C09107=1044.224,228.789,397.774,171.384,39.330,157.455
C09108=1044.218,228.541,397.802,171.382,39.328,157.454
C09109=1044.211,228.292,397.829,171.380,39.325,157.454
C09110=1044.204,228.044,397.856,171.378,39.323,157.453
C09111=1044.197,227.795,397.883,171.375,39.321,157.453
C09112=1044.191,227.547,397.911,171.373,39.319,157.452
C09113=1044.184,227.299,397.939,171.370,39.316,157.452
C09114=1044.178,227.051,397.966,171.369,39.314,157.451
C09115=1044.171,226.802,397.994,171.366,39.312,157.451
C09116=1044.164,226.554,398.022,171.364,39.309,157.450
C09117=1044.158,226.305,398.049,171.361,39.306,157.449
C09118=1044.151,226.056,398.076,171.358,39.304,157.449
C09119=1044.145,225.809,398.103,171.357,39.302,157.448
C09120=1044.138,225.560,398.131,171.354,39.299,157.448
C09121=1044.131,225.312,398.159,171.352,39.297,157.447
C09122=1044.125,225.063,398.186,171.349,39.295,157.446
C09123=1044.118,224.814,398.213,171.347,39.292,157.446
C09124=1044.111,224.566,398.241,171.345,39.290,157.445
C09125=1044.106,224.318,398.268,171.343,39.287,157.445
C09126=1044.099,224.069,398.296,171.340,39.285,157.444
C09127=1044.092,223.821,398.323,171.337,39.283,157.444
C09128=1044.085,223.573,398.350,171.336,39.280,157.443
C09129=1044.079,223.324,398.377,171.333,39.277,157.442
C09130=1044.072,223.076,398.405,171.331,39.275,157.442
C09131=1044.066,222.827,398.433,171.328,39.273,157.441
C09132=1044.059,222.578,398.460,171.327,39.271,157.441
C09133=1044.053,222.331,398.487,171.324,39.268,157.440
C09134=1044.046,222.082,398.514,171.322,39.266,157.440
C09135=1044.040,221.833,398.541,171.319,39.263,157.439
C09136=1044.033,221.585,398.569,171.317,39.261,157.438
C09137=1044.027,221.337,398.595,171.315,39.258,157.438
C09138=1044.019,221.044,398.628,171.312,39.255,157.437
C09139=1044.012,220.752,398.660,171.310,39.253,157.436
C09140=1044.003,220.459,398.692,171.307,39.250,157.436
C09141=1043.996,220.167,398.724,171.304,39.247,157.435
C09142=1043.990,219.918,398.751,171.302,39.244,157.434
C09143=1043.983,219.670,398.778,171.299,39.242,157.434
C09144=1043.976,219.421,398.805,171.298,39.240,157.433
C09145=1043.969,219.173,398.832,171.295,39.237,157.433
C09146=1043.963,218.925,398.859,171.293,39.235,157.432
C09147=1043.956,218.676,398.886,171.290,39.233,157.432
C09148=1043.950,218.428,398.913,171.288,39.230,157.431
C09149=1043.943,218.179,398.940,171.286,39.228,157.430
C09150=1043.936,217.930,398.966,171.283,39.225,157.430
C09151=1043.929,217.682,398.994,171.282,39.223,157.429
C09152=1043.924,217.433,399.021,171.279,39.221,157.429
C09153=1043.916,217.185,399.048,171.277,39.218,157.428
C09154=1043.910,216.936,399.075,171.275,39.216,157.428
C09155=1043.903,216.688,399.101,171.273,39.213,157.427
C09156=1043.897,216.440,399.129,171.270,39.211,157.426
C09157=1043.890,216.191,399.155,171.268,39.208,157.426
C09158=1043.884,215.943,399.182,171.266,39.206,157.425
C09159=1043.877,215.694,399.210,171.263,39.204,157.425
C09160=1043.870,215.445,399.236,171.261,39.201,157.424
C09161=1043.864,215.197,399.263,171.259,39.199,157.424
C09162=1043.857,214.949,399.290,171.257,39.196,157.423
C09163=1043.851,214.701,399.316,171.254,39.194,157.422
C09164=1043.844,214.452,399.343,171.253,39.191,157.422
C09165=1043.838,214.203,399.370,171.250,39.189,157.421
C09166=1043.829,213.866,399.406,171.247,39.186,157.420
C09167=1043.820,213.528,399.442,171.245,39.182,157.420
C09168=1043.811,213.191,399.479,171.241,39.179,157.419
C09169=1043.802,212.853,399.515,171.238,39.176,157.418
C09170=1043.796,212.606,399.542,171.237,39.173,157.418
C09171=1043.789,212.357,399.569,171.234,39.171,157.417
C09172=1043.782,212.108,399.596,171.231,39.168,157.416
C09173=1043.777,211.860,399.622,171.230,39.166,157.416
C09174=1043.769,211.611,399.649,171.227,39.163,157.415
C09175=1043.763,211.363,399.675,171.226,39.161,157.415
C09176=1043.757,211.114,399.702,171.223,39.159,157.414
C09177=1043.750,210.866,399.729,171.221,39.156,157.414
C09178=1043.743,210.617,399.756,171.219,39.153,157.413
C09179=1043.736,210.368,399.782,171.217,39.151,157.412
C09180=1043.730,210.120,399.808,171.214,39.149,157.412
C09181=1043.723,209.871,399.835,171.213,39.146,157.411
C09182=1043.717,209.623,399.861,171.210,39.144,157.411
C09183=1043.710,209.374,399.888,171.208,39.141,157.410
C09184=1043.704,209.126,399.914,171.206,39.139,157.409
C09185=1043.697,208.877,399.941,171.203,39.137,157.409
C09186=1043.690,208.629,399.967,171.202,39.134,157.408
C09187=1043.684,208.380,399.994,171.199,39.132,157.408
C09188=1043.677,208.132,400.020,171.198,39.129,157.407
C09189=1043.670,207.883,400.046,171.195,39.127,157.407
C09190=1043.665,207.660,400.071,171.194,39.125,157.406
C09191=1043.659,207.437,400.094,171.191,39.122,157.406
C09192=1043.653,207.214,400.117,171.190,39.120,157.405
C09193=1043.646,206.990,400.141,171.187,39.118,157.405
C09194=1043.641,206.767,400.164,171.186,39.116,157.404
C09195=1043.635,206.544,400.188,171.184,39.114,157.404
C09196=1043.628,206.321,400.212,171.182,39.111,157.403
C09197=1043.623,206.097,400.236,171.181,39.110,157.403
C09198=1043.597,205.046,400.342,170.913,39.008,157.374
C09199=1043.591,204.797,400.367,170.910,39.006,157.373
C09200=1043.585,204.548,400.392,170.907,39.004,157.373
C09201=1043.578,204.300,400.417,170.905,39.003,157.373
C09202=1043.572,204.051,400.442,170.901,39.001,157.372
C09203=1043.566,203.802,400.468,170.899,38.999,157.372
C09204=1043.560,203.554,400.493,170.895,38.998,157.371
C09205=1043.554,203.305,400.517,170.893,38.996,157.371
C09206=1043.548,203.056,400.543,170.890,38.994,157.370
C09207=1043.542,202.808,400.568,170.887,38.993,157.370
C09208=1043.536,202.559,400.593,170.884,38.991,157.370
C09209=1043.530,202.310,400.618,170.882,38.989,157.369
C09210=1043.524,202.062,400.643,170.879,38.987,157.369
C09211=1043.518,201.813,400.668,170.876,38.986,157.368
C09212=1043.512,201.565,400.694,170.873,38.984,157.368
C09213=1043.506,201.315,400.718,170.870,38.982,157.368
C09214=1043.499,201.067,400.743,170.868,38.981,157.367
C09215=1043.493,200.818,400.768,170.864,38.979,157.367
C09216=1043.487,200.570,400.792,170.862,38.978,157.366
C09217=1043.480,200.321,400.817,170.859,38.976,157.366
C09218=1043.474,200.072,400.842,170.856,38.975,157.366
C09219=1043.468,199.824,400.867,170.853,38.973,157.365
C09220=1043.462,199.574,400.891,170.851,38.972,157.365
C09221=1043.455,199.326,400.916,170.848,38.970,157.364
C09222=1043.449,199.077,400.940,170.845,38.968,157.364
C09223=1043.443,198.829,400.966,170.842,38.967,157.364
C09224=1043.437,198.580,400.990,170.839,38.966,157.363
C09225=1043.430,198.331,401.015,170.837,38.964,157.363
C09226=1043.424,198.082,401.039,170.833,38.962,157.362
C09227=1043.418,197.834,401.064,170.831,38.961,157.362
C09228=1043.411,197.585,401.088,170.828,38.960,157.362
C09229=1043.405,197.336,401.113,170.825,38.958,157.361
C09230=1043.399,197.087,401.138,170.823,38.956,157.361
C09231=1043.393,196.840,401.162,170.820,38.954,157.360
C09232=1043.387,196.590,401.187,170.817,38.953,157.360
C09233=1043.380,196.341,401.211,170.814,38.952,157.360
C09234=1043.374,196.093,401.236,170.812,38.950,157.359
C09235=1043.368,195.844,401.260,170.809,38.949,157.359
C09236=1043.362,195.596,401.285,170.806,38.947,157.359
C09237=1043.356,195.346,401.310,170.804,38.945,157.358
C09238=1043.350,195.098,401.334,170.800,38.944,157.358
C09239=1043.344,194.849,401.359,170.798,38.943,157.357
C09240=1043.337,194.600,401.383,170.795,38.941,157.357
C09241=1043.331,194.351,401.408,170.792,38.939,157.357
C09242=1043.325,194.104,401.432,170.790,38.938,157.356
C09243=1043.319,193.854,401.457,170.786,38.937,157.356
C09244=1043.312,193.605,401.481,170.784,38.935,157.355
C09245=1043.307,193.357,401.506,170.782,38.934,157.355
C09246=1043.301,193.108,401.530,170.778,38.932,157.355
C09247=1043.295,192.860,401.554,170.776,38.930,157.354
C09248=1043.289,192.610,401.579,170.774,38.929,157.354
C09249=1043.282,192.362,401.603,170.770,38.928,157.354
C09250=1043.277,192.113,401.628,170.768,38.926,157.353
C09251=1043.270,191.864,401.652,170.765,38.925,157.353
C09252=1043.264,191.615,401.676,170.762,38.923,157.352
C09253=1043.258,191.367,401.700,170.760,38.921,157.352
C09254=1043.252,191.118,401.725,170.757,38.920,157.352
C09255=1043.246,190.870,401.749,170.754,38.919,157.351
C09256=1043.240,190.621,401.774,170.752,38.917,157.351
C09257=1043.233,190.372,401.798,170.749,38.916,157.351
C09258=1043.228,190.123,401.822,170.746,38.914,157.350
C09259=1043.221,189.839,401.850,170.743,38.912,157.350
C09260=1043.214,189.554,401.877,170.741,38.911,157.349
C09261=1043.207,189.271,401.905,170.737,38.909,157.349
C09262=1043.201,188.985,401.933,170.734,38.907,157.349
C09263=1043.194,188.736,401.957,170.732,38.906,157.348
C09264=1043.189,188.488,401.981,170.729,38.905,157.348
C09265=1043.182,188.239,402.005,170.727,38.903,157.347
C09266=1043.176,187.991,402.030,170.724,38.902,157.347
C09267=1043.170,187.742,402.054,170.721,38.900,157.347
C09268=1043.165,187.493,402.078,170.719,38.899,157.346
C09269=1043.158,187.244,402.103,170.716,38.897,157.346
C09270=1043.153,186.996,402.127,170.713,38.895,157.346
C09271=1043.146,186.747,402.151,170.711,38.894,157.345
C09272=1043.141,186.498,402.175,170.708,38.893,157.345
C09273=1043.134,186.249,402.199,170.705,38.892,157.345
C09274=1043.129,186.001,402.223,170.703,38.890,157.344
C09275=1043.123,185.752,402.247,170.701,38.888,157.344
C09276=1043.117,185.503,402.272,170.697,38.887,157.343
C09277=1043.111,185.255,402.295,170.695,38.885,157.343
C09278=1043.104,185.005,402.319,170.693,38.884,157.343
C09279=1043.099,184.757,402.343,170.690,38.882,157.342
C09280=1043.092,184.508,402.367,170.687,38.881,157.342
C09281=1043.087,184.259,402.391,170.685,38.880,157.342
C09282=1043.081,184.010,402.415,170.682,38.878,157.341
C09283=1043.075,183.761,402.439,170.680,38.877,157.341
C09284=1043.069,183.513,402.463,170.677,38.875,157.340
C09285=1043.063,183.264,402.486,170.674,38.874,157.340
C09286=1043.056,183.015,402.510,170.672,38.873,157.340
C09287=1043.050,182.766,402.534,170.669,38.872,157.340
C09288=1043.044,182.517,402.558,170.666,38.870,157.339
C09289=1043.038,182.268,402.581,170.664,38.869,157.339
C09290=1043.031,182.019,402.605,170.661,38.868,157.339
C09291=1043.024,181.771,402.628,170.659,38.866,157.338
C09292=1043.018,181.522,402.651,170.656,38.865,157.338
C09293=1043.012,181.274,402.675,170.653,38.864,157.338
C09294=1043.005,181.025,402.699,170.651,38.863,157.337
C09295=1043.000,180.776,402.722,170.648,38.861,157.337
C09296=1042.993,180.527,402.746,170.646,38.860,157.337
C09297=1042.987,180.278,402.770,170.643,38.859,157.336
C09298=1042.981,180.030,402.793,170.641,38.858,157.336
C09299=1042.975,179.781,402.817,170.638,38.856,157.336
C09300=1042.969,179.532,402.840,170.635,38.855,157.335
C09301=1042.962,179.283,402.864,170.633,38.854,157.335
C09302=1042.957,179.034,402.887,170.631,38.853,157.335
C09303=1042.949,178.785,402.910,170.628,38.851,157.334
C09304=1042.943,178.537,402.934,170.625,38.850,157.334
C09305=1042.937,178.288,402.957,170.623,38.849,157.334
C09306=1042.931,178.039,402.981,170.620,38.848,157.334
C09307=1042.925,177.790,403.004,170.618,38.846,157.333
C09308=1042.918,177.541,403.028,170.615,38.845,157.333
C09309=1042.913,177.292,403.051,170.613,38.844,157.333
C09310=1042.907,177.044,403.074,170.610,38.843,157.332
C09311=1042.900,176.794,403.098,170.608,38.841,157.332
C09312=1042.894,176.546,403.121,170.605,38.840,157.332
C09313=1042.887,176.297,403.144,170.602,38.839,157.331
C09314=1042.881,176.049,403.168,170.600,38.838,157.331
C09315=1042.875,175.800,403.191,170.598,38.837,157.331
C09316=1042.869,175.550,403.214,170.596,38.835,157.330
C09317=1042.863,175.302,403.238,170.592,38.834,157.330
C09318=1042.857,175.053,403.261,170.590,38.833,157.330
C09319=1042.851,174.804,403.285,170.588,38.832,157.329
C09320=1042.845,174.555,403.308,170.586,38.831,157.329
C09321=1042.838,174.306,403.330,170.582,38.829,157.329
C09322=1042.832,174.057,403.354,170.580,38.828,157.328
C09323=1042.826,173.773,403.380,170.578,38.827,157.328
C09324=1042.818,173.488,403.407,170.574,38.825,157.328
C09325=1042.811,173.203,403.434,170.572,38.823,157.327
C09326=1042.805,172.918,403.461,170.569,38.822,157.327
C09327=1042.799,172.670,403.484,170.566,38.821,157.327
C09328=1042.792,172.420,403.506,170.564,38.820,157.326
C09329=1042.786,172.171,403.529,170.562,38.818,157.326
C09330=1042.780,171.923,403.553,170.559,38.817,157.326
C09331=1042.774,171.674,403.576,170.556,38.816,157.325
C09332=1042.768,171.425,403.599,170.554,38.815,157.325
C09333=1042.762,171.176,403.623,170.552,38.814,157.325
C09334=1042.756,170.928,403.645,170.549,38.812,157.324
C09335=1042.750,170.679,403.668,170.547,38.811,157.324
C09336=1042.743,170.429,403.691,170.544,38.810,157.324
C09337=1042.737,170.181,403.715,170.542,38.809,157.324
C09338=1042.732,169.932,403.738,170.539,38.808,157.323
C09339=1042.726,169.683,403.761,170.537,38.806,157.323
C09340=1042.720,169.434,403.784,170.535,38.805,157.323
C09341=1042.713,169.185,403.807,170.533,38.804,157.322
C09342=1042.707,168.937,403.830,170.529,38.803,157.322
C09343=1042.701,168.688,403.853,170.527,38.801,157.322
C09344=1042.696,168.439,403.876,170.525,38.800,157.321
C09345=1042.690,168.190,403.899,170.522,38.799,157.321
C09346=1042.683,167.941,403.922,170.520,38.797,157.321
C09347=1042.677,167.692,403.945,170.518,38.796,157.321
C09348=1042.671,167.443,403.968,170.516,38.795,157.320
C09349=1042.665,167.195,403.991,170.512,38.794,157.320
C09350=1042.660,166.946,404.014,170.510,38.792,157.320
C09351=1042.654,166.697,404.037,170.508,38.791,157.319
C09352=1042.647,166.448,404.060,170.506,38.790,157.319
C09353=1042.641,166.199,404.083,170.503,38.789,157.319
C09354=1042.635,165.950,404.106,170.501,38.788,157.318
C09355=1042.630,165.701,404.129,170.499,38.787,157.318
C09356=1042.624,165.452,404.152,170.496,38.785,157.318
C09357=1042.617,165.203,404.174,170.494,38.784,157.317
C09358=1042.612,164.955,404.197,170.491,38.783,157.317
C09359=1042.606,164.706,404.220,170.489,38.782,157.317
C09360=1042.600,164.457,404.243,170.486,38.781,157.317
C09361=1042.595,164.208,404.266,170.484,38.779,157.316
C09362=1042.588,163.959,404.288,170.482,38.778,157.316
C09363=1042.582,163.710,404.311,170.480,38.777,157.316
C09364=1042.577,163.461,404.334,170.477,38.775,157.315
C09365=1042.570,163.212,404.357,170.475,38.774,157.315
C09366=1042.565,162.963,404.380,170.473,38.773,157.315
C09367=1042.558,162.714,404.403,170.471,38.772,157.314
C09368=1042.552,162.466,404.426,170.467,38.770,157.314
C09369=1042.547,162.217,404.449,170.465,38.769,157.314
C09370=1042.541,161.968,404.472,170.463,38.768,157.313
C09371=1042.535,161.719,404.495,170.460,38.767,157.313
C09372=1042.529,161.470,404.517,170.458,38.766,157.313
C09373=1042.523,161.221,404.540,170.456,38.765,157.313
C09374=1042.517,160.972,404.563,170.454,38.763,157.312
C09375=1042.512,160.723,404.585,170.451,38.762,157.312
C09376=1042.505,160.474,404.607,170.449,38.761,157.312
C09377=1042.500,160.225,404.630,170.447,38.760,157.311
C09378=1042.494,159.977,404.653,170.445,38.758,157.311
C09379=1042.487,159.728,404.676,170.442,38.757,157.311
C09380=1042.481,159.479,404.697,170.440,38.756,157.311
C09381=1042.475,159.230,404.720,170.437,38.755,157.310
C09382=1042.469,158.981,404.743,170.435,38.754,157.310
C09383=1042.463,158.732,404.764,170.432,38.753,157.310
C09384=1042.457,158.483,404.787,170.430,38.752,157.309
C09385=1042.451,158.235,404.809,170.428,38.751,157.309
C09386=1042.445,157.986,404.832,170.426,38.749,157.309
C09387=1042.438,157.700,404.858,170.423,38.748,157.309
C09388=1042.431,157.414,404.883,170.420,38.747,157.308
C09389=1042.424,157.130,404.909,170.418,38.746,157.308
C09390=1042.417,156.844,404.934,170.416,38.745,157.308
C09391=1042.411,156.595,404.957,170.412,38.744,157.307
C09392=1042.404,156.346,404.979,170.410,38.743,157.307
C09393=1042.398,156.097,405.001,170.408,38.742,157.307
C09394=1042.392,155.848,405.024,170.406,38.741,157.307
C09395=1042.386,155.599,405.046,170.403,38.739,157.306
C09396=1042.380,155.350,405.068,170.401,38.738,157.306
C09397=1042.374,155.102,405.091,170.399,38.737,157.306
C09398=1042.368,154.852,405.113,170.397,38.736,157.305
C09399=1042.361,154.604,405.135,170.394,38.735,157.305
C09400=1042.356,154.354,405.157,170.392,38.734,157.305
C09401=1042.350,154.106,405.179,170.390,38.733,157.305
C09402=1042.343,153.856,405.201,170.388,38.732,157.304
C09403=1042.337,153.608,405.223,170.386,38.731,157.304
C09404=1042.331,153.358,405.246,170.383,38.730,157.304
C09405=1042.325,153.110,405.268,170.381,38.729,157.304
C09406=1042.319,152.861,405.290,170.379,38.728,157.303
C09407=1042.312,152.612,405.312,170.377,38.726,157.303
C09408=1042.307,152.364,405.333,170.373,38.725,157.303
C09409=1042.301,152.115,405.356,170.371,38.724,157.302
C09410=1042.295,151.865,405.378,170.369,38.724,157.302
C09411=1042.288,151.617,405.400,170.367,38.723,157.302
C09412=1042.282,151.368,405.422,170.364,38.721,157.302
C09413=1042.277,151.118,405.444,170.362,38.720,157.302
C09414=1042.270,150.870,405.466,170.360,38.719,157.301
C09415=1042.264,150.620,405.488,170.358,38.718,157.301
C09416=1042.258,150.372,405.510,170.355,38.717,157.301
C09417=1042.252,150.123,405.532,170.353,38.716,157.300
C09418=1042.246,149.873,405.554,170.351,38.715,157.300
C09419=1042.240,149.624,405.577,170.349,38.714,157.300
C09420=1042.234,149.376,405.598,170.347,38.713,157.300
C09421=1042.228,149.127,405.620,170.344,38.712,157.299
C09422=1042.222,148.878,405.642,170.342,38.711,157.299
C09423=1042.215,148.629,405.664,170.340,38.710,157.299
C09424=1042.209,148.380,405.685,170.338,38.709,157.299
C09425=1042.203,148.131,405.708,170.335,38.708,157.298
C09426=1042.197,147.882,405.730,170.333,38.707,157.298
C09427=1042.191,147.632,405.751,170.331,38.706,157.298
C09428=1042.186,147.384,405.773,170.329,38.705,157.298
C09429=1042.179,147.135,405.795,170.326,38.703,157.297
C09430=1042.173,146.886,405.817,170.324,38.703,157.297
C09431=1042.167,146.637,405.838,170.322,38.702,157.297
C09432=1042.161,146.388,405.860,170.320,38.701,157.297
C09433=1042.154,146.138,405.882,170.318,38.699,157.296
C09434=1042.148,145.890,405.904,170.315,38.699,157.296
C09435=1042.142,145.641,405.925,170.313,38.698,157.296
C09436=1042.136,145.392,405.947,170.311,38.697,157.296
C09437=1042.130,145.143,405.968,170.309,38.696,157.295
C09438=1042.124,144.894,405.990,170.307,38.695,157.295
C09439=1042.118,144.645,406.012,170.304,38.694,157.295
C09440=1042.111,144.396,406.034,170.302,38.693,157.295
C09441=1042.106,144.147,406.055,170.300,38.692,157.294
C09442=1042.099,143.899,406.076,170.298,38.691,157.294
C09443=1042.093,143.649,406.098,170.296,38.690,157.294
C09444=1042.087,143.400,406.120,170.293,38.689,157.294
C09445=1042.080,143.151,406.141,170.291,38.688,157.293
C09446=1042.074,142.902,406.163,170.289,38.687,157.293
C09447=1042.069,142.653,406.184,170.287,38.686,157.293
C09448=1042.062,142.404,406.206,170.284,38.685,157.293
C09449=1042.056,142.155,406.227,170.282,38.684,157.292
C09450=1042.050,141.906,406.249,170.280,38.683,157.292
C09451=1042.044,141.621,406.274,170.278,38.682,157.292
C09452=1042.036,141.335,406.299,170.275,38.681,157.292
C09453=1042.029,141.049,406.323,170.272,38.680,157.291
C09454=1042.022,140.764,406.348,170.270,38.679,157.291
C09455=1042.017,140.515,406.370,170.268,38.678,157.291
C09456=1042.010,140.266,406.391,170.266,38.677,157.291
C09457=1042.004,140.017,406.413,170.263,38.676,157.290
C09458=1041.997,139.768,406.434,170.261,38.675,157.290
C09459=1041.992,139.519,406.455,170.259,38.674,157.290
C09460=1041.986,139.270,406.477,170.257,38.673,157.290
C09461=1041.980,139.021,406.498,170.255,38.672,157.289
C09462=1041.974,138.771,406.519,170.252,38.671,157.289
C09463=1041.968,138.523,406.541,170.250,38.670,157.289
C09464=1041.961,138.274,406.562,170.248,38.669,157.289
C09465=1041.955,138.024,406.583,170.246,38.668,157.288
C09466=1041.949,137.775,406.605,170.244,38.667,157.288
C09467=1041.943,137.527,406.626,170.241,38.666,157.288
C09468=1041.936,137.278,406.647,170.239,38.665,157.288
C09469=1041.930,137.029,406.669,170.237,38.664,157.287
C09470=1041.924,136.779,406.690,170.235,38.664,157.287
C09471=1041.918,136.531,406.711,170.233,38.663,157.287
C09472=1041.912,136.281,406.732,170.230,38.661,157.287
C09473=1041.906,136.032,406.754,170.229,38.661,157.287
C09474=1041.900,135.784,406.775,170.227,38.660,157.286
C09475=1041.894,135.534,406.795,170.225,38.659,157.286
C09476=1041.887,135.285,406.817,170.223,38.658,157.286
C09477=1041.882,135.036,406.838,170.220,38.657,157.286
C09478=1041.875,134.788,406.859,170.218,38.656,157.285
C09479=1041.869,134.538,406.880,170.216,38.655,157.285
C09480=1041.864,134.289,406.902,170.214,38.654,157.285
C09481=1041.857,134.040,406.923,170.211,38.653,157.285
C09482=1041.851,133.791,406.944,170.209,38.652,157.284
C09483=1041.845,133.542,406.965,170.207,38.651,157.284
C09484=1041.838,133.293,406.986,170.205,38.651,157.284
C09485=1041.832,133.044,407.007,170.203,38.650,157.284
C09486=1041.827,132.795,407.029,170.200,38.648,157.283
C09487=1041.820,132.546,407.049,170.198,38.648,157.283
C09488=1041.814,132.297,407.071,170.196,38.647,157.283
C09489=1041.808,132.048,407.092,170.194,38.646,157.283
C09490=1041.802,131.799,407.112,170.193,38.645,157.283
C09491=1041.796,131.550,407.134,170.191,38.644,157.282
C09492=1041.790,131.301,407.155,170.188,38.643,157.282
C09493=1041.783,131.051,407.175,170.186,38.642,157.282
C09494=1041.778,130.803,407.197,170.184,38.641,157.282
C09495=1041.771,130.553,407.217,170.182,38.641,157.281
C09496=1041.764,130.305,407.238,170.180,38.640,157.281
C09497=1041.759,130.055,407.259,170.177,38.639,157.281
C09498=1041.752,129.807,407.280,170.175,38.638,157.281
C09499=1041.746,129.557,407.300,170.173,38.637,157.281
C09500=1041.740,129.309,407.321,170.171,38.636,157.280
C09501=1041.733,129.059,407.342,170.169,38.636,157.280
C09502=1041.727,128.810,407.363,170.166,38.635,157.280
C09503=1041.721,128.561,407.383,170.164,38.634,157.280
C09504=1041.714,128.312,407.404,170.162,38.633,157.279
C09505=1041.708,128.063,407.425,170.160,38.632,157.279
C09506=1041.702,127.814,407.446,170.158,38.631,157.279
C09507=1041.696,127.565,407.466,170.157,38.631,157.279
C09508=1041.690,127.316,407.487,170.154,38.629,157.279
C09509=1041.683,127.067,407.508,170.152,38.629,157.278
C09510=1041.677,126.818,407.529,170.150,38.628,157.278
C09511=1041.671,126.569,407.549,170.148,38.627,157.278
C09512=1041.665,126.319,407.570,170.146,38.626,157.278
C09513=1041.658,126.071,407.590,170.143,38.626,157.278
C09514=1041.653,125.821,407.611,170.141,38.625,157.277
C09515=1041.646,125.536,407.635,170.139,38.623,157.277
C09516=1041.638,125.249,407.659,170.137,38.623,157.277
C09517=1041.631,124.964,407.683,170.134,38.622,157.277
C09518=1041.624,124.678,407.706,170.131,38.621,157.276
C09519=1041.617,124.429,407.727,170.129,38.620,157.276
C09520=1041.611,124.179,407.748,170.127,38.619,157.276
C09521=1041.605,123.931,407.767,170.126,38.618,157.276
C09522=1041.599,123.682,407.789,170.124,38.617,157.276
C09523=1041.593,123.433,407.809,170.122,38.617,157.275
C09524=1041.587,123.183,407.829,170.119,38.616,157.275
C09525=1041.580,122.935,407.850,170.117,38.615,157.275
C09526=1041.574,122.685,407.870,170.115,38.614,157.275
C09527=1041.569,122.436,407.891,170.113,38.613,157.274
C09528=1041.562,122.187,407.912,170.111,38.612,157.274
C09529=1041.556,121.938,407.932,170.108,38.611,157.274
C09530=1041.550,121.689,407.953,170.106,38.611,157.274
C09531=1041.544,121.440,407.973,170.105,38.609,157.274
C09532=1041.537,121.191,407.994,170.103,38.609,157.273
C09533=1041.532,120.942,408.014,170.101,38.608,157.273
C09534=1041.525,120.692,408.035,170.098,38.607,157.273
C09535=1041.519,120.443,408.055,170.096,38.606,157.273
C09536=1041.514,120.195,408.076,170.094,38.605,157.273
C09537=1041.507,119.945,408.096,170.092,38.604,157.272
C09538=1041.501,119.697,408.116,170.090,38.604,157.272
C09539=1041.494,119.447,408.137,170.089,38.603,157.272
C09540=1041.489,119.199,408.158,170.086,38.601,157.272
C09541=1041.482,118.949,408.178,170.084,38.601,157.271
C09542=1041.476,118.700,408.198,170.082,38.600,157.271
C09543=1041.470,118.450,408.219,170.080,38.599,157.271
C09544=1041.464,118.202,408.239,170.078,38.598,157.271
C09545=1041.458,117.953,408.259,170.075,38.598,157.271
C09546=1041.451,117.704,408.280,170.073,38.596,157.270
C09547=1041.446,117.455,408.301,170.072,38.596,157.270
C09548=1041.440,117.205,408.321,170.070,38.595,157.270
C09549=1041.434,116.956,408.341,170.068,38.594,157.270
C09550=1041.428,116.707,408.361,170.065,38.593,157.269
C09551=1041.422,116.458,408.382,170.063,38.592,157.269
C09552=1041.416,116.209,408.402,170.061,38.591,157.269
C09553=1041.410,115.960,408.422,170.059,38.590,157.269
C09554=1041.404,115.710,408.443,170.058,38.590,157.269
C09555=1041.398,115.462,408.463,170.055,38.589,157.268
C09556=1041.391,115.213,408.484,170.053,38.588,157.268
C09557=1041.385,114.964,408.504,170.051,38.587,157.268
C09558=1041.380,114.715,408.524,170.049,38.586,157.268
C09559=1041.373,114.465,408.544,170.047,38.585,157.267
C09560=1041.367,114.216,408.564,170.046,38.584,157.267
C09561=1041.362,113.967,408.585,170.043,38.583,157.267
C09562=1041.355,113.718,408.605,170.041,38.582,157.267
C09563=1041.349,113.469,408.625,170.039,38.582,157.267
C09564=1041.343,113.220,408.645,170.037,38.581,157.266
C09565=1041.337,112.971,408.665,170.035,38.580,157.266
C09566=1041.331,112.722,408.685,170.032,38.579,157.266
C09567=1041.325,112.473,408.705,170.031,38.578,157.266
C09568=1041.318,112.224,408.726,170.029,38.577,157.266
C09569=1041.312,111.975,408.746,170.027,38.577,157.265
C09570=1041.306,111.725,408.765,170.025,38.576,157.265
C09571=1041.300,111.476,408.785,170.023,38.575,157.265
C09572=1041.294,111.227,408.805,170.020,38.574,157.265
C09573=1041.287,110.977,408.826,170.018,38.573,157.265
C09574=1041.281,110.729,408.846,170.017,38.573,157.264
C09575=1041.275,110.480,408.865,170.015,38.572,157.264
C09576=1041.269,110.230,408.886,170.013,38.571,157.264
C09577=1041.263,109.981,408.905,170.011,38.571,157.264
C09578=1041.257,109.732,408.925,170.008,38.569,157.264
C09579=1041.249,109.421,408.950,170.006,38.568,157.263
C09580=1041.241,109.110,408.974,170.003,38.568,157.263
C09581=1041.233,108.799,408.999,170.001,38.567,157.263
C09582=1041.226,108.489,409.024,169.999,38.565,157.263
C09583=1041.220,108.252,409.043,169.996,38.565,157.262
C09584=1041.213,108.015,409.062,169.994,38.564,157.262
C09585=1041.208,107.779,409.081,169.992,38.563,157.262
C09586=1041.202,107.542,409.099,169.991,38.563,157.262
C09587=1041.196,107.305,409.118,169.989,38.562,157.262
C09588=1041.189,107.068,409.137,169.987,38.561,157.261
C09589=1041.184,106.832,409.156,169.984,38.561,157.261
C09590=1041.178,106.595,409.174,169.983,38.560,157.261
C09591=1041.172,106.346,409.194,169.981,38.559,157.261
C09592=1041.166,106.097,409.214,169.979,38.558,157.261
C09593=1041.160,105.848,409.234,169.977,38.558,157.261
C09594=1041.153,105.598,409.254,169.975,38.557,157.260
C09595=1041.147,105.349,409.274,169.973,38.556,157.260
C09596=1041.141,105.101,409.293,169.971,38.555,157.260
C09597=1041.134,104.851,409.312,169.969,38.554,157.260
C09598=1041.128,104.602,409.332,169.967,38.554,157.260
C09599=1041.122,104.353,409.352,169.965,38.553,157.259
C09600=1041.117,104.104,409.372,169.963,38.552,157.259
C09601=1041.111,103.855,409.392,169.960,38.551,157.259
C09602=1041.104,103.605,409.411,169.959,38.550,157.259
C09603=1041.098,103.356,409.431,169.957,38.550,157.259
C09604=1041.092,103.107,409.451,169.955,38.549,157.258
C09605=1041.086,102.858,409.470,169.953,38.548,157.258
C09606=1041.079,102.608,409.490,169.951,38.547,157.258
C09607=1041.073,102.359,409.509,169.948,38.546,157.258
C09608=1041.067,102.110,409.529,169.947,38.546,157.258
C09609=1041.061,101.862,409.549,169.945,38.545,157.257
C09610=1041.055,101.612,409.568,169.943,38.544,157.257
C09611=1041.049,101.363,409.588,169.941,38.543,157.257
C09612=1041.042,101.114,409.607,169.939,38.543,157.257
C09613=1041.036,100.865,409.627,169.936,38.541,157.257
C09614=1041.030,100.615,409.646,169.935,38.541,157.256
C09615=1041.024,100.366,409.666,169.933,38.540,157.256
C09616=1041.017,100.117,409.685,169.931,38.539,157.256
C09617=1041.011,99.868,409.705,169.929,38.539,157.256
C09618=1041.005,99.619,409.724,169.927,38.538,157.256
C09619=1040.999,99.370,409.744,169.924,38.537,157.255
C09620=1040.993,99.120,409.763,169.923,38.536,157.255
C09621=1040.986,98.871,409.783,169.921,38.536,157.255
C09622=1040.980,98.622,409.802,169.919,38.535,157.255
C09623=1040.974,98.373,409.821,169.917,38.534,157.255
C09624=1040.968,98.124,409.840,169.915,38.534,157.255
C09625=1040.961,97.875,409.859,169.913,38.533,157.254
C09626=1040.955,97.625,409.879,169.911,38.532,157.254
C09627=1040.948,97.376,409.898,169.909,38.531,157.254
C09628=1040.943,97.127,409.917,169.907,38.531,157.254
C09629=1040.936,96.878,409.937,169.905,38.530,157.254
C09630=1040.930,96.629,409.956,169.903,38.529,157.253
C09631=1040.924,96.380,409.975,169.901,38.529,157.253
C09632=1040.917,96.130,409.995,169.899,38.527,157.253
C09633=1040.912,95.881,410.014,169.897,38.527,157.253
C09634=1040.905,95.632,410.033,169.895,38.526,157.253
C09635=1040.899,95.383,410.053,169.893,38.525,157.252
C09636=1040.893,95.134,410.071,169.891,38.525,157.252
C09637=1040.887,94.884,410.091,169.889,38.524,157.252
C09638=1040.880,94.636,410.110,169.887,38.523,157.252
C09639=1040.875,94.386,410.129,169.885,38.522,157.252
C09640=1040.868,94.136,410.148,169.883,38.522,157.252
C09641=1040.862,93.888,410.168,169.881,38.521,157.251
C09642=1040.855,93.639,410.187,169.879,38.520,157.251
C09643=1040.848,93.352,410.209,169.877,38.520,157.251
C09644=1040.841,93.066,410.231,169.874,38.518,157.251
C09645=1040.835,92.781,410.253,169.872,38.518,157.251
C09646=1040.827,92.495,410.275,169.870,38.517,157.250
C09647=1040.821,92.246,410.294,169.868,38.516,157.250
C09648=1040.815,91.996,410.313,169.866,38.515,157.250
C09649=1040.808,91.746,410.332,169.864,38.515,157.250
C09650=1040.802,91.498,410.352,169.863,38.514,157.250
C09651=1040.796,91.249,410.371,169.860,38.513,157.249
C09652=1040.790,90.999,410.390,169.858,38.512,157.249
C09653=1040.784,90.750,410.408,169.856,38.512,157.249
C09654=1040.778,90.501,410.428,169.854,38.511,157.249
C09655=1040.772,90.251,410.446,169.853,38.510,157.249
C09656=1040.766,90.003,410.466,169.851,38.509,157.248
C09657=1040.759,89.754,410.485,169.848,38.508,157.248
C09658=1040.753,89.504,410.504,169.846,38.508,157.248
C09659=1040.746,89.255,410.522,169.844,38.507,157.248
C09660=1040.741,89.006,410.542,169.842,38.507,157.248
C09661=1040.734,88.757,410.560,169.841,38.506,157.247
C09662=1040.728,88.508,410.579,169.839,38.505,157.247
C09663=1040.721,88.258,410.598,169.837,38.504,157.247
C09664=1040.715,88.008,410.617,169.834,38.504,157.247
C09665=1040.709,87.759,410.636,169.832,38.503,157.247
C09666=1040.702,87.510,410.654,169.830,38.502,157.247
C09667=1040.696,87.261,410.673,169.829,38.502,157.246
C09668=1040.690,87.012,410.692,169.827,38.501,157.246
C09669=1040.684,86.762,410.711,169.825,38.501,157.246
C09670=1040.677,86.513,410.730,169.822,38.499,157.246
C09671=1040.671,86.264,410.748,169.820,38.499,157.246
C09672=1040.664,86.015,410.767,169.818,38.498,157.246
C09673=1040.659,85.766,410.786,169.817,38.498,157.245
C09674=1040.652,85.516,410.805,169.815,38.497,157.245
C09675=1040.646,85.267,410.823,169.813,38.496,157.245
C09676=1040.639,85.018,410.842,169.811,38.496,157.245
C09677=1040.633,84.769,410.861,169.808,38.495,157.245
C09678=1040.627,84.520,410.880,169.807,38.494,157.245
C09679=1040.621,84.271,410.899,169.805,38.493,157.244
C09680=1040.615,84.021,410.917,169.803,38.493,157.244
C09681=1040.608,83.772,410.936,169.801,38.492,157.244
C09682=1040.602,83.523,410.955,169.799,38.492,157.244
C09683=1040.596,83.274,410.974,169.797,38.491,157.244
C09684=1040.590,83.025,410.992,169.795,38.490,157.243
C09685=1040.583,82.775,411.010,169.793,38.489,157.243
C09686=1040.577,82.526,411.029,169.791,38.488,157.243
C09687=1040.571,82.276,411.048,169.789,38.488,157.243
C09688=1040.565,82.027,411.067,169.787,38.487,157.243
C09689=1040.558,81.778,411.086,169.786,38.487,157.243
C09690=1040.552,81.529,411.104,169.783,38.485,157.242
C09691=1040.546,81.281,411.122,169.781,38.485,157.242
C09692=1040.540,81.031,411.140,169.779,38.484,157.242
C09693=1040.534,80.781,411.160,169.777,38.484,157.242
C09694=1040.528,80.532,411.178,169.775,38.483,157.242
C09695=1040.522,80.283,411.197,169.774,38.482,157.242
C09696=1040.515,80.034,411.216,169.772,38.482,157.241
C09697=1040.509,79.785,411.234,169.769,38.480,157.241
C09698=1040.503,79.535,411.253,169.767,38.480,157.241
C09699=1040.497,79.286,411.271,169.765,38.479,157.241
C09700=1040.490,79.037,411.290,169.764,38.479,157.241
C09701=1040.485,78.788,411.308,169.762,38.478,157.240
C09702=1040.479,78.538,411.326,169.760,38.477,157.240
C09703=1040.472,78.289,411.345,169.758,38.477,157.240
C09704=1040.466,78.040,411.364,169.755,38.476,157.240
C09705=1040.459,77.791,411.382,169.754,38.475,157.240
C09706=1040.453,77.541,411.400,169.752,38.474,157.240
C09707=1040.446,77.255,411.422,169.750,38.474,157.239
C09708=1040.439,76.969,411.443,169.748,38.473,157.239
C09709=1040.432,76.683,411.464,169.746,38.472,157.239
C09710=1040.424,76.397,411.486,169.742,38.472,157.239
C09711=1040.418,76.147,411.504,169.741,38.470,157.239
C09712=1040.413,75.899,411.522,169.739,38.470,157.238
C09713=1040.406,75.649,411.539,169.737,38.469,157.238
C09714=1040.399,75.400,411.558,169.735,38.469,157.238
C09715=1040.393,75.151,411.577,169.733,38.468,157.238
C09716=1040.387,74.901,411.594,169.731,38.468,157.238
C09717=1040.380,74.652,411.613,169.729,38.466,157.238
C09718=1040.374,74.403,411.631,169.727,38.466,157.237
C09719=1040.368,74.153,411.650,169.725,38.465,157.237
C09720=1040.362,73.905,411.668,169.723,38.465,157.237
C09721=1040.356,73.655,411.686,169.721,38.464,157.237
C09722=1040.349,73.406,411.705,169.719,38.463,157.237
C09723=1040.343,73.156,411.723,169.718,38.463,157.237
C09724=1040.337,72.907,411.741,169.715,38.462,157.236
C09725=1040.330,72.658,411.759,169.713,38.461,157.236
C09726=1040.324,72.410,411.777,169.711,38.461,157.236
C09727=1040.318,72.160,411.795,169.709,38.460,157.236
C09728=1040.312,71.911,411.813,169.708,38.459,157.236
C09729=1040.305,71.662,411.832,169.706,38.459,157.236
C09730=1040.299,71.412,411.850,169.704,38.458,157.235
C09731=1040.293,71.163,411.868,169.702,38.458,157.235
C09732=1040.287,70.914,411.886,169.699,38.457,157.235
C09733=1040.280,70.664,411.904,169.697,38.456,157.235
C09734=1040.274,70.415,411.922,169.696,38.455,157.235
C09735=1040.268,70.165,411.940,169.694,38.455,157.235
C09736=1040.262,69.917,411.958,169.692,38.454,157.234
C09737=1040.256,69.667,411.976,169.690,38.454,157.234
C09738=1040.249,69.418,411.995,169.687,38.453,157.234
C09739=1040.243,69.168,412.013,169.686,38.452,157.234
C09740=1040.236,68.919,412.031,169.684,38.451,157.234
C09741=1040.230,68.670,412.049,169.682,38.451,157.234
C09742=1040.224,68.421,412.066,169.680,38.450,157.233
C09743=1040.218,68.172,412.085,169.678,38.450,157.233
C09744=1040.211,67.922,412.102,169.676,38.449,157.233
C09745=1040.205,67.672,412.120,169.675,38.448,157.233
C09746=1040.199,67.424,412.139,169.672,38.447,157.233
C09747=1040.193,67.174,412.157,169.670,38.447,157.233
C09748=1040.186,66.925,412.174,169.668,38.446,157.232
C09749=1040.180,66.676,412.193,169.666,38.446,157.232
C09750=1040.174,66.427,412.210,169.664,38.445,157.232
C09751=1040.167,66.177,412.227,169.663,38.444,157.232
C09752=1040.161,65.928,412.246,169.661,38.444,157.232
C09753=1040.155,65.678,412.264,169.658,38.443,157.232
C09754=1040.149,65.430,412.281,169.656,38.443,157.231
C09755=1040.142,65.181,412.300,169.654,38.442,157.231
C09756=1040.136,64.931,412.318,169.652,38.441,157.231
C09757=1040.129,64.681,412.335,169.651,38.441,157.231
C09758=1040.124,64.432,412.353,169.649,38.440,157.231
C09759=1040.117,64.183,412.371,169.647,38.439,157.231
C09760=1040.110,63.934,412.388,169.644,38.439,157.230
C09761=1040.104,63.684,412.406,169.642,38.438,157.230
C09762=1040.098,63.435,412.423,169.640,38.438,157.230
C09763=1040.092,63.186,412.441,169.639,38.437,157.230
C09764=1040.085,62.936,412.459,169.637,38.436,157.230
C09765=1040.079,62.687,412.477,169.635,38.436,157.230
C09766=1040.072,62.438,412.494,169.633,38.435,157.230
C09767=1040.065,62.189,412.512,169.631,38.435,157.229
C09768=1040.059,61.939,412.530,169.629,38.434,157.229
C09769=1040.052,61.690,412.547,169.626,38.434,157.229
C09770=1040.047,61.441,412.564,169.624,38.433,157.229
C09771=1040.039,61.154,412.585,169.622,38.433,157.229
C09772=1040.032,60.868,412.604,169.620,38.432,157.229
C09773=1040.024,60.582,412.624,169.618,38.432,157.229
C09774=1040.017,60.296,412.644,169.616,38.431,157.228
C09775=1040.011,60.047,412.663,169.614,38.431,157.228
C09776=1040.004,59.797,412.680,169.612,38.430,157.228
C09777=1039.998,59.547,412.698,169.609,38.429,157.228
C09778=1039.991,59.299,412.715,169.607,38.428,157.228
C09779=1039.985,59.049,412.733,169.606,38.428,157.228
C09780=1039.979,58.800,412.751,169.604,38.427,157.227
C09781=1039.972,58.551,412.768,169.602,38.427,157.227
C09782=1039.965,58.301,412.785,169.600,38.426,157.227
C09783=1039.959,58.052,412.803,169.598,38.426,157.227
C09784=1039.953,57.803,412.820,169.595,38.425,157.227
C09785=1039.947,57.553,412.838,169.593,38.424,157.227
C09786=1039.940,57.304,412.855,169.592,38.424,157.227
C09787=1039.934,57.055,412.872,169.590,38.423,157.226
C09788=1039.928,56.805,412.890,169.588,38.423,157.226
C09789=1039.921,56.556,412.907,169.586,38.422,157.226
C09790=1039.915,56.307,412.924,169.584,38.422,157.226
C09791=1039.908,56.057,412.942,169.582,38.421,157.226
C09792=1039.902,55.809,412.959,169.580,38.421,157.226
C09793=1039.896,55.559,412.977,169.578,38.420,157.226
C09794=1039.889,55.310,412.994,169.576,38.420,157.225
C09795=1039.883,55.060,413.011,169.574,38.419,157.225
C09796=1039.877,54.810,413.029,169.572,38.418,157.225
C09797=1039.871,54.562,413.046,169.570,38.418,157.225
C09798=1039.864,54.312,413.063,169.568,38.417,157.225
C09799=1039.858,54.063,413.081,169.566,38.417,157.225
C09800=1039.852,53.814,413.098,169.565,38.416,157.225
C09801=1039.845,53.564,413.115,169.562,38.415,157.224
C09802=1039.839,53.315,413.133,169.560,38.415,157.224
C09803=1039.832,53.066,413.150,169.558,38.414,157.224
C09804=1039.827,52.816,413.167,169.556,38.413,157.224
C09805=1039.820,52.567,413.184,169.554,38.413,157.224
C09806=1039.813,52.317,413.202,169.552,38.412,157.224
C09807=1039.808,52.068,413.219,169.551,38.412,157.223
C09808=1039.801,51.819,413.237,169.549,38.411,157.223
C09809=1039.795,51.570,413.254,169.546,38.411,157.223
C09810=1039.789,51.320,413.271,169.544,38.410,157.223
C09811=1039.783,51.071,413.288,169.542,38.410,157.223
C09812=1039.776,50.822,413.305,169.540,38.409,157.223
C09813=1039.770,50.573,413.323,169.539,38.409,157.223
C09814=1039.764,50.323,413.340,169.537,38.407,157.222
C09815=1039.758,50.074,413.356,169.535,38.407,157.222
C09816=1039.751,49.824,413.374,169.532,38.406,157.222
C09817=1039.745,49.575,413.391,169.530,38.406,157.222
C09818=1039.738,49.326,413.408,169.528,38.405,157.222
C09819=1039.733,49.077,413.426,169.526,38.405,157.222
C09820=1039.726,48.827,413.443,169.525,38.404,157.221
C09821=1039.720,48.578,413.460,169.523,38.403,157.221
C09822=1039.714,48.328,413.478,169.521,38.403,157.221
C09823=1039.708,48.079,413.494,169.519,38.402,157.221
C09824=1039.701,47.830,413.511,169.516,38.401,157.221
C09825=1039.696,47.581,413.529,169.514,38.401,157.221
C09826=1039.689,47.331,413.546,169.512,38.400,157.220
C09827=1039.683,47.082,413.562,169.511,38.400,157.220
C09828=1039.676,46.832,413.580,169.509,38.399,157.220
C09829=1039.670,46.583,413.597,169.507,38.398,157.220
C09830=1039.664,46.333,413.614,169.505,38.398,157.220
C09831=1039.658,46.085,413.631,169.503,38.397,157.220
C09832=1039.652,45.835,413.648,169.500,38.397,157.220
C09833=1039.646,45.585,413.665,169.499,38.396,157.219
C09834=1039.639,45.337,413.682,169.497,38.395,157.219
C09835=1039.632,45.049,413.702,169.495,38.395,157.219
C09836=1039.625,44.764,413.722,169.492,38.394,157.219
C09837=1039.618,44.477,413.741,169.490,38.393,157.219
C09838=1039.611,44.190,413.760,169.488,38.392,157.218
C09839=1039.605,43.941,413.777,169.485,38.392,157.218
C09840=1039.598,43.692,413.795,169.484,38.391,157.218
C09841=1039.593,43.442,413.812,169.482,38.391,157.218
C09842=1039.587,43.193,413.828,169.480,38.390,157.218
C09843=1039.580,42.943,413.845,169.478,38.390,157.218
C09844=1039.574,42.694,413.862,169.476,38.389,157.218
C09845=1039.567,42.444,413.879,169.474,38.388,157.217
C09846=1039.561,42.196,413.896,169.472,38.388,157.217
C09847=1039.554,41.946,413.912,169.469,38.387,157.217
C09848=1039.548,41.697,413.929,169.468,38.387,157.217
C09849=1039.542,41.447,413.946,169.466,38.386,157.217
C09850=1039.535,41.198,413.963,169.464,38.386,157.217
C09851=1039.529,40.949,413.979,169.462,38.385,157.217
C09852=1039.522,40.699,413.996,169.460,38.385,157.216
C09853=1039.517,40.450,414.013,169.458,38.384,157.216
C09854=1039.511,40.200,414.030,169.456,38.384,157.216
C09855=1039.504,39.951,414.047,169.454,38.383,157.216
C09856=1039.499,39.701,414.063,169.451,38.382,157.216
C09857=1039.492,39.452,414.080,169.450,38.381,157.216
C09858=1039.486,39.203,414.097,169.448,38.381,157.215
C09859=1039.479,38.954,414.114,169.446,38.380,157.215
C09860=1039.473,38.704,414.130,169.444,38.380,157.215
C09861=1039.467,38.455,414.147,169.442,38.379,157.215
C09862=1039.461,38.206,414.164,169.440,38.379,157.215
C09863=1039.454,37.956,414.180,169.437,38.378,157.215
C09864=1039.448,37.706,414.196,169.435,38.377,157.215
C09865=1039.442,37.458,414.213,169.433,38.377,157.214
C09866=1039.435,37.208,414.230,169.432,38.376,157.214
C09867=1039.429,36.958,414.246,169.430,38.376,157.214
C09868=1039.422,36.710,414.263,169.428,38.376,157.214
C09869=1039.416,36.460,414.279,169.426,38.375,157.214
C09870=1039.410,36.210,414.296,169.424,38.375,157.214
C09871=1039.403,35.960,414.312,169.422,38.374,157.214
C09872=1039.397,35.712,414.329,169.420,38.374,157.214
C09873=1039.391,35.462,414.345,169.417,38.373,157.213
C09874=1039.384,35.213,414.361,169.415,38.373,157.213
C09875=1039.378,34.963,414.378,169.413,38.372,157.213
C09876=1039.372,34.715,414.395,169.411,38.372,157.213
C09877=1039.365,34.464,414.411,169.410,38.371,157.213
C09878=1039.359,34.215,414.428,169.408,38.370,157.213
C09879=1039.352,33.966,414.443,169.406,38.370,157.213
C09880=1039.346,33.717,414.461,169.404,38.370,157.212
C09881=1039.340,33.467,414.477,169.402,38.369,157.212
C09882=1039.334,33.218,414.493,169.399,38.369,157.212
C09883=1039.328,32.969,414.509,169.397,38.368,157.212
C09884=1039.320,32.719,414.525,169.395,38.368,157.212
C09885=1039.315,32.470,414.542,169.393,38.367,157.212
C09886=1039.308,32.221,414.559,169.391,38.367,157.212
C09887=1039.302,31.971,414.575,169.389,38.366,157.211
C09888=1039.295,31.722,414.591,169.387,38.366,157.211
C09889=1039.289,31.472,414.607,169.385,38.365,157.211
C09890=1039.283,31.223,414.623,169.383,38.364,157.211
C09891=1039.277,30.973,414.640,169.381,38.364,157.211
C09892=1039.271,30.724,414.656,169.379,38.363,157.211
C09893=1039.264,30.475,414.673,169.377,38.363,157.211
C09894=1039.258,30.226,414.689,169.375,38.363,157.211
C09895=1039.251,29.976,414.706,169.373,38.362,157.210
C09896=1039.245,29.726,414.722,169.371,38.362,157.210
C09897=1039.238,29.477,414.737,169.369,38.361,157.210
C09898=1039.233,29.228,414.754,169.367,38.361,157.210
C09899=1039.225,28.941,414.773,169.365,38.360,157.210
C09900=1039.218,28.654,414.791,169.362,38.360,157.210
C09901=1039.211,28.368,414.810,169.360,38.358,157.209
C09902=1039.203,28.081,414.828,169.357,38.358,157.209
C09903=1039.197,27.832,414.845,169.355,38.358,157.209
C09904=1039.190,27.582,414.861,169.353,38.358,157.209
C09905=1039.184,27.333,414.877,169.352,38.357,157.209
C09906=1039.178,27.084,414.893,169.350,38.356,157.209
C09907=1039.172,26.834,414.908,169.348,38.356,157.209
C09908=1039.166,26.585,414.924,169.345,38.355,157.209
C09909=1039.159,26.335,414.941,169.343,38.355,157.208
C09910=1039.153,26.086,414.957,169.341,38.355,157.208
C09911=1039.147,25.836,414.973,169.339,38.354,157.208
C09912=1039.140,25.587,414.989,169.337,38.354,157.208
C09913=1039.133,25.337,415.005,169.335,38.353,157.208
C09914=1039.127,25.088,415.021,169.333,38.353,157.208
C09915=1039.121,24.839,415.037,169.331,38.352,157.208
C09916=1039.114,24.590,415.053,169.329,38.352,157.208
C09917=1039.108,24.340,415.069,169.327,38.352,157.208
C09918=1039.103,24.090,415.085,169.324,38.351,157.207
C09919=1039.095,23.841,415.101,169.322,38.351,157.207
C09920=1039.089,23.591,415.117,169.320,38.350,157.207
C09921=1039.083,23.342,415.133,169.318,38.349,157.207
C09922=1039.077,23.093,415.149,169.316,38.349,157.207
C09923=1039.070,22.844,415.165,169.314,38.349,157.207
C09924=1039.064,22.595,415.181,169.312,38.348,157.207
C09925=1039.057,22.344,415.196,169.310,38.348,157.206
C09926=1039.051,22.095,415.212,169.308,38.347,157.206
C09927=1039.044,21.846,415.228,169.307,38.347,157.206
C09928=1039.038,21.596,415.244,169.304,38.346,157.206
C09929=1039.032,21.347,415.260,169.302,38.346,157.206
C09930=1039.026,21.097,415.276,169.300,38.345,157.206
C09931=1039.019,20.848,415.291,169.298,38.345,157.206
C09932=1039.013,20.599,415.307,169.296,38.345,157.206
C09933=1039.007,20.350,415.323,169.294,38.344,157.205
C09934=1039.001,20.099,415.339,169.292,38.344,157.205
C09935=1038.994,19.850,415.355,169.290,38.343,157.205
C09936=1038.988,19.601,415.371,169.288,38.342,157.205
C09937=1038.981,19.352,415.387,169.286,38.343,157.205
C09938=1038.976,19.102,415.402,169.283,38.342,157.205
C09939=1038.969,18.853,415.418,169.281,38.342,157.205
C09940=1038.962,18.604,415.433,169.279,38.341,157.205
C09941=1038.957,18.354,415.449,169.277,38.340,157.204
C09942=1038.950,18.105,415.465,169.275,38.341,157.204
C09943=1038.944,17.856,415.481,169.273,38.340,157.204
C09944=1038.937,17.605,415.496,169.271,38.339,157.204
C09945=1038.930,17.356,415.512,169.269,38.339,157.204
C09946=1038.924,17.107,415.528,169.267,38.338,157.204
C09947=1038.918,16.857,415.543,169.265,38.338,157.204
C09948=1038.911,16.608,415.559,169.262,38.338,157.204
C09949=1038.906,16.358,415.574,169.260,38.337,157.203
C09950=1038.899,16.109,415.590,169.258,38.337,157.203
C09951=1038.893,15.860,415.606,169.256,38.336,157.203
C09952=1038.887,15.610,415.621,169.254,38.336,157.203
C09953=1038.880,15.361,415.637,169.252,38.336,157.203
C09954=1038.874,15.111,415.652,169.250,38.335,157.203
C09955=1038.868,14.862,415.668,169.248,38.335,157.203
C09956=1038.861,14.612,415.683,169.246,38.334,157.203
C09957=1038.855,14.363,415.699,169.244,38.334,157.202
C09958=1038.848,14.114,415.715,169.242,38.334,157.202
C09959=1038.842,13.864,415.730,169.239,38.333,157.202
C09960=1038.836,13.615,415.745,169.237,38.333,157.202
C09961=1038.830,13.365,415.761,169.235,38.332,157.202
C09962=1038.823,13.116,415.776,169.233,38.332,157.202
C09963=1038.816,12.830,415.794,169.231,38.332,157.202
C09964=1038.808,12.545,415.811,169.228,38.331,157.202
C09965=1038.801,12.260,415.829,169.226,38.331,157.202
C09966=1038.794,11.974,415.846,169.224,38.331,157.202
C09967=1038.787,11.725,415.862,169.222,38.330,157.201
C09968=1038.780,11.475,415.877,169.220,38.330,157.201
C09969=1038.774,11.226,415.892,169.218,38.330,157.201
C09970=1038.768,10.976,415.908,169.215,38.329,157.201
C09971=1038.762,10.727,415.923,169.213,38.329,157.201
C09972=1038.755,10.478,415.938,169.210,38.329,157.201
C09973=1038.749,10.228,415.953,169.208,38.328,157.201
C09974=1038.742,9.979,415.969,169.206,38.328,157.201
C09975=1038.736,9.729,415.984,169.204,38.328,157.201
C09976=1038.729,9.480,415.999,169.202,38.327,157.200
C09977=1038.723,9.231,416.015,169.200,38.327,157.200
C09978=1038.716,8.981,416.029,169.198,38.327,157.200
C09979=1038.710,8.731,416.044,169.196,38.326,157.200
C09980=1038.704,8.482,416.061,169.194,38.326,157.200
C09981=1038.697,8.232,416.076,169.191,38.325,157.200
C09982=1038.691,7.983,416.091,169.189,38.325,157.200
C09983=1038.684,7.734,416.106,169.187,38.325,157.200
C09984=1038.678,7.484,416.121,169.185,38.324,157.200
C09985=1038.672,7.234,416.136,169.183,38.324,157.199
C09986=1038.665,6.985,416.151,169.181,38.324,157.199
C09987=1038.659,6.736,416.167,169.179,38.323,157.199
C09988=1038.652,6.486,416.182,169.177,38.323,157.199
C09989=1038.646,6.237,416.196,169.175,38.323,157.199
C09990=1038.640,5.987,416.211,169.173,38.322,157.199
C09991=1038.633,5.738,416.227,169.171,38.321,157.199
C09992=1038.627,5.489,416.242,169.169,38.322,157.199
C09993=1038.621,5.239,416.257,169.166,38.321,157.199
C09994=1038.615,4.989,416.272,169.163,38.320,157.198
C09995=1038.608,4.739,416.287,169.161,38.321,157.198
C09996=1038.602,4.490,416.303,169.159,38.320,157.198
//INST
///DATE 2021/06/25 14:48
///ATTR SC,RW,RJ
////FRAME ROBOT
///GROUP1 RB1
NOP
MOVL C00000 V=800.0 PL=0
MOVL C00001 V=800.0 PL=0
MOVL C00002 V=800.0 PL=0
MOVL C00003 V=800.0 PL=0
MOVL C00004 V=800.0 PL=0
MOVL C00005 V=800.0 PL=0
MOVL C00006 V=800.0 PL=0
MOVL C00007 V=800.0 PL=0
MOVL C00008 V=800.0 PL=0
MOVL C00009 V=800.0 PL=0
MOVL C00010 V=800.0 PL=0
MOVL C00011 V=800.0 PL=0
MOVL C00012 V=800.0 PL=0
MOVL C00013 V=800.0 PL=0
MOVL C00014 V=800.0 PL=0
MOVL C00015 V=800.0 PL=0
MOVL C00016 V=800.0 PL=0
MOVL C00017 V=800.0 PL=0
MOVL C00018 V=800.0 PL=0
MOVL C00019 V=800.0 PL=0
MOVL C00020 V=800.0 PL=0
MOVL C00021 V=800.0 PL=0
MOVL C00022 V=800.0 PL=0
MOVL C00023 V=800.0 PL=0
MOVL C00024 V=800.0 PL=0
MOVL C00025 V=800.0 PL=0
MOVL C00026 V=800.0 PL=0
MOVL C00027 V=800.0 PL=0
MOVL C00028 V=800.0 PL=0
MOVL C00029 V=800.0 PL=0
MOVL C00030 V=800.0 PL=0
MOVL C00031 V=800.0 PL=0
MOVL C00032 V=800.0 PL=0
MOVL C00033 V=800.0 PL=0
MOVL C00034 V=800.0 PL=0
MOVL C00035 V=800.0 PL=0
MOVL C00036 V=800.0 PL=0
MOVL C00037 V=800.0 PL=0
MOVL C00038 V=800.0 PL=0
MOVL C00039 V=800.0 PL=0
MOVL C00040 V=800.0 PL=0
MOVL C00041 V=800.0 PL=0
MOVL C00042 V=800.0 PL=0
MOVL C00043 V=800.0 PL=0
MOVL C00044 V=800.0 PL=0
MOVL C00045 V=800.0 PL=0
MOVL C00046 V=800.0 PL=0
MOVL C00047 V=800.0 PL=0
MOVL C00048 V=800.0 PL=0
MOVL C00049 V=800.0 PL=0
MOVL C00050 V=800.0 PL=0
MOVL C00051 V=800.0 PL=0
MOVL C00052 V=800.0 PL=0
MOVL C00053 V=800.0 PL=0
MOVL C00054 V=800.0 PL=0
MOVL C00055 V=800.0 PL=0
MOVL C00056 V=800.0 PL=0
MOVL C00057 V=800.0 PL=0
MOVL C00058 V=800.0 PL=0
MOVL C00059 V=800.0 PL=0
MOVL C00060 V=800.0 PL=0
MOVL C00061 V=800.0 PL=0
MOVL C00062 V=800.0 PL=0
MOVL C00063 V=800.0 PL=0
MOVL C00064 V=800.0 PL=0
MOVL C00065 V=800.0 PL=0
MOVL C00066 V=800.0 PL=0
MOVL C00067 V=800.0 PL=0
MOVL C00068 V=800.0 PL=0
MOVL C00069 V=800.0 PL=0
MOVL C00070 V=800.0 PL=0
MOVL C00071 V=800.0 PL=0
MOVL C00072 V=800.0 PL=0
MOVL C00073 V=800.0 PL=0
MOVL C00074 V=800.0 PL=0
MOVL C00075 V=800.0 PL=0
MOVL C00076 V=800.0 PL=0
MOVL C00077 V=800.0 PL=0
MOVL C00078 V=800.0 PL=0
MOVL C00079 V=800.0 PL=0
MOVL C00080 V=800.0 PL=0
MOVL C00081 V=800.0 PL=0
MOVL C00082 V=800.0 PL=0
MOVL C00083 V=800.0 PL=0
MOVL C00084 V=800.0 PL=0
MOVL C00085 V=800.0 PL=0
MOVL C00086 V=800.0 PL=0
MOVL C00087 V=800.0 PL=0
MOVL C00088 V=800.0 PL=0
MOVL C00089 V=800.0 PL=0
MOVL C00090 V=800.0 PL=0
MOVL C00091 V=800.0 PL=0
MOVL C00092 V=800.0 PL=0
MOVL C00093 V=800.0 PL=0
MOVL C00094 V=800.0 PL=0
MOVL C00095 V=800.0 PL=0
MOVL C00096 V=800.0 PL=0
MOVL C00097 V=800.0 PL=0
MOVL C00098 V=800.0 PL=0
MOVL C00099 V=800.0 PL=0
MOVL C00100 V=800.0 PL=0
MOVL C00101 V=800.0 PL=0
MOVL C00102 V=800.0 PL=0
MOVL C00103 V=800.0 PL=0
MOVL C00104 V=800.0 PL=0
MOVL C00105 V=800.0 PL=0
MOVL C00106 V=800.0 PL=0
MOVL C00107 V=800.0 PL=0
MOVL C00108 V=800.0 PL=0
MOVL C00109 V=800.0 PL=0
MOVL C00110 V=800.0 PL=0
MOVL C00111 V=800.0 PL=0
MOVL C00112 V=800.0 PL=0
MOVL C00113 V=800.0 PL=0
MOVL C00114 V=800.0 PL=0
MOVL C00115 V=800.0 PL=0
MOVL C00116 V=800.0 PL=0
MOVL C00117 V=800.0 PL=0
MOVL C00118 V=800.0 PL=0
MOVL C00119 V=800.0 PL=0
MOVL C00120 V=800.0 PL=0
MOVL C00121 V=800.0 PL=0
MOVL C00122 V=800.0 PL=0
MOVL C00123 V=800.0 PL=0
MOVL C00124 V=800.0 PL=0
MOVL C00125 V=800.0 PL=0
MOVL C00126 V=800.0 PL=0
MOVL C00127 V=800.0 PL=0
MOVL C00128 V=800.0 PL=0
MOVL C00129 V=800.0 PL=0
MOVL C00130 V=800.0 PL=0
MOVL C00131 V=800.0 PL=0
MOVL C00132 V=800.0 PL=0
MOVL C00133 V=800.0 PL=0
MOVL C00134 V=800.0 PL=0
MOVL C00135 V=800.0 PL=0
MOVL C00136 V=800.0 PL=0
MOVL C00137 V=800.0 PL=0
MOVL C00138 V=800.0 PL=0
MOVL C00139 V=800.0 PL=0
MOVL C00140 V=800.0 PL=0
MOVL C00141 V=800.0 PL=0
MOVL C00142 V=800.0 PL=0
MOVL C00143 V=800.0 PL=0
MOVL C00144 V=800.0 PL=0
MOVL C00145 V=800.0 PL=0
MOVL C00146 V=800.0 PL=0
MOVL C00147 V=800.0 PL=0
MOVL C00148 V=800.0 PL=0
MOVL C00149 V=800.0 PL=0
MOVL C00150 V=800.0 PL=0
MOVL C00151 V=800.0 PL=0
MOVL C00152 V=800.0 PL=0
MOVL C00153 V=800.0 PL=0
MOVL C00154 V=800.0 PL=0
MOVL C00155 V=800.0 PL=0
MOVL C00156 V=800.0 PL=0
MOVL C00157 V=800.0 PL=0
MOVL C00158 V=800.0 PL=0
MOVL C00159 V=800.0 PL=0
MOVL C00160 V=800.0 PL=0
MOVL C00161 V=800.0 PL=0
MOVL C00162 V=800.0 PL=0
MOVL C00163 V=800.0 PL=0
MOVL C00164 V=800.0 PL=0
MOVL C00165 V=800.0 PL=0
MOVL C00166 V=800.0 PL=0
MOVL C00167 V=800.0 PL=0
MOVL C00168 V=800.0 PL=0
MOVL C00169 V=800.0 PL=0
MOVL C00170 V=800.0 PL=0
MOVL C00171 V=800.0 PL=0
MOVL C00172 V=800.0 PL=0
MOVL C00173 V=800.0 PL=0
MOVL C00174 V=800.0 PL=0
MOVL C00175 V=800.0 PL=0
MOVL C00176 V=800.0 PL=0
MOVL C00177 V=800.0 PL=0
MOVL C00178 V=800.0 PL=0
MOVL C00179 V=800.0 PL=0
MOVL C00180 V=800.0 PL=0
MOVL C00181 V=800.0 PL=0
MOVL C00182 V=800.0 PL=0
MOVL C00183 V=800.0 PL=0
MOVL C00184 V=800.0 PL=0
MOVL C00185 V=800.0 PL=0
MOVL C00186 V=800.0 PL=0
MOVL C00187 V=800.0 PL=0
MOVL C00188 V=800.0 PL=0
MOVL C00189 V=800.0 PL=0
MOVL C00190 V=800.0 PL=0
MOVL C00191 V=800.0 PL=0
MOVL C00192 V=800.0 PL=0
MOVL C00193 V=800.0 PL=0
MOVL C00194 V=800.0 PL=0
MOVL C00195 V=800.0 PL=0
MOVL C00196 V=800.0 PL=0
MOVL C00197 V=800.0 PL=0
MOVL C00198 V=800.0 PL=0
MOVL C00199 V=800.0 PL=0
MOVL C00200 V=800.0 PL=0
MOVL C00201 V=800.0 PL=0
MOVL C00202 V=800.0 PL=0
MOVL C00203 V=800.0 PL=0
MOVL C00204 V=800.0 PL=0
MOVL C00205 V=800.0 PL=0
MOVL C00206 V=800.0 PL=0
MOVL C00207 V=800.0 PL=0
MOVL C00208 V=800.0 PL=0
MOVL C00209 V=800.0 PL=0
MOVL C00210 V=800.0 PL=0
MOVL C00211 V=800.0 PL=0
MOVL C00212 V=800.0 PL=0
MOVL C00213 V=800.0 PL=0
MOVL C00214 V=800.0 PL=0
MOVL C00215 V=800.0 PL=0
MOVL C00216 V=800.0 PL=0
MOVL C00217 V=800.0 PL=0
MOVL C00218 V=800.0 PL=0
MOVL C00219 V=800.0 PL=0
MOVL C00220 V=800.0 PL=0
MOVL C00221 V=800.0 PL=0
MOVL C00222 V=800.0 PL=0
MOVL C00223 V=800.0 PL=0
MOVL C00224 V=800.0 PL=0
MOVL C00225 V=800.0 PL=0
MOVL C00226 V=800.0 PL=0
MOVL C00227 V=800.0 PL=0
MOVL C00228 V=800.0 PL=0
MOVL C00229 V=800.0 PL=0
MOVL C00230 V=800.0 PL=0
MOVL C00231 V=800.0 PL=0
MOVL C00232 V=800.0 PL=0
MOVL C00233 V=800.0 PL=0
MOVL C00234 V=800.0 PL=0
MOVL C00235 V=800.0 PL=0
MOVL C00236 V=800.0 PL=0
MOVL C00237 V=800.0 PL=0
MOVL C00238 V=800.0 PL=0
MOVL C00239 V=800.0 PL=0
MOVL C00240 V=800.0 PL=0
MOVL C00241 V=800.0 PL=0
MOVL C00242 V=800.0 PL=0
MOVL C00243 V=800.0 PL=0
MOVL C00244 V=800.0 PL=0
MOVL C00245 V=800.0 PL=0
MOVL C00246 V=800.0 PL=0
MOVL C00247 V=800.0 PL=0
MOVL C00248 V=800.0 PL=0
MOVL C00249 V=800.0 PL=0
MOVL C00250 V=800.0 PL=0
MOVL C00251 V=800.0 PL=0
MOVL C00252 V=800.0 PL=0
MOVL C00253 V=800.0 PL=0
MOVL C00254 V=800.0 PL=0
MOVL C00255 V=800.0 PL=0
MOVL C00256 V=800.0 PL=0
MOVL C00257 V=800.0 PL=0
MOVL C00258 V=800.0 PL=0
MOVL C00259 V=800.0 PL=0
MOVL C00260 V=800.0 PL=0
MOVL C00261 V=800.0 PL=0
MOVL C00262 V=800.0 PL=0
MOVL C00263 V=800.0 PL=0
MOVL C00264 V=800.0 PL=0
MOVL C00265 V=800.0 PL=0
MOVL C00266 V=800.0 PL=0
MOVL C00267 V=800.0 PL=0
MOVL C00268 V=800.0 PL=0
MOVL C00269 V=800.0 PL=0
MOVL C00270 V=800.0 PL=0
MOVL C00271 V=800.0 PL=0
MOVL C00272 V=800.0 PL=0
MOVL C00273 V=800.0 PL=0
MOVL C00274 V=800.0 PL=0
MOVL C00275 V=800.0 PL=0
MOVL C00276 V=800.0 PL=0
MOVL C00277 V=800.0 PL=0
MOVL C00278 V=800.0 PL=0
MOVL C00279 V=800.0 PL=0
MOVL C00280 V=800.0 PL=0
MOVL C00281 V=800.0 PL=0
MOVL C00282 V=800.0 PL=0
MOVL C00283 V=800.0 PL=0
MOVL C00284 V=800.0 PL=0
MOVL C00285 V=800.0 PL=0
MOVL C00286 V=800.0 PL=0
MOVL C00287 V=800.0 PL=0
MOVL C00288 V=800.0 PL=0
MOVL C00289 V=800.0 PL=0
MOVL C00290 V=800.0 PL=0
MOVL C00291 V=800.0 PL=0
MOVL C00292 V=800.0 PL=0
MOVL C00293 V=800.0 PL=0
MOVL C00294 V=800.0 PL=0
MOVL C00295 V=800.0 PL=0
MOVL C00296 V=800.0 PL=0
MOVL C00297 V=800.0 PL=0
MOVL C00298 V=800.0 PL=0
MOVL C00299 V=800.0 PL=0
MOVL C00300 V=800.0 PL=0
MOVL C00301 V=800.0 PL=0
MOVL C00302 V=800.0 PL=0
MOVL C00303 V=800.0 PL=0
MOVL C00304 V=800.0 PL=0
MOVL C00305 V=800.0 PL=0
MOVL C00306 V=800.0 PL=0
MOVL C00307 V=800.0 PL=0
MOVL C00308 V=800.0 PL=0
MOVL C00309 V=800.0 PL=0
MOVL C00310 V=800.0 PL=0
MOVL C00311 V=800.0 PL=0
MOVL C00312 V=800.0 PL=0
MOVL C00313 V=800.0 PL=0
MOVL C00314 V=800.0 PL=0
MOVL C00315 V=800.0 PL=0
MOVL C00316 V=800.0 PL=0
MOVL C00317 V=800.0 PL=0
MOVL C00318 V=800.0 PL=0
MOVL C00319 V=800.0 PL=0
MOVL C00320 V=800.0 PL=0
MOVL C00321 V=800.0 PL=0
MOVL C00322 V=800.0 PL=0
MOVL C00323 V=800.0 PL=0
MOVL C00324 V=800.0 PL=0
MOVL C00325 V=800.0 PL=0
MOVL C00326 V=800.0 PL=0
MOVL C00327 V=800.0 PL=0
MOVL C00328 V=800.0 PL=0
MOVL C00329 V=800.0 PL=0
MOVL C00330 V=800.0 PL=0
MOVL C00331 V=800.0 PL=0
MOVL C00332 V=800.0 PL=0
MOVL C00333 V=800.0 PL=0
MOVL C00334 V=800.0 PL=0
MOVL C00335 V=800.0 PL=0
MOVL C00336 V=800.0 PL=0
MOVL C00337 V=800.0 PL=0
MOVL C00338 V=800.0 PL=0
MOVL C00339 V=800.0 PL=0
MOVL C00340 V=800.0 PL=0
MOVL C00341 V=800.0 PL=0
MOVL C00342 V=800.0 PL=0
MOVL C00343 V=800.0 PL=0
MOVL C00344 V=800.0 PL=0
MOVL C00345 V=800.0 PL=0
MOVL C00346 V=800.0 PL=0
MOVL C00347 V=800.0 PL=0
MOVL C00348 V=800.0 PL=0
MOVL C00349 V=800.0 PL=0
MOVL C00350 V=800.0 PL=0
MOVL C00351 V=800.0 PL=0
MOVL C00352 V=800.0 PL=0
MOVL C00353 V=800.0 PL=0
MOVL C00354 V=800.0 PL=0
MOVL C00355 V=800.0 PL=0
MOVL C00356 V=800.0 PL=0
MOVL C00357 V=800.0 PL=0
MOVL C00358 V=800.0 PL=0
MOVL C00359 V=800.0 PL=0
MOVL C00360 V=800.0 PL=0
MOVL C00361 V=800.0 PL=0
MOVL C00362 V=800.0 PL=0
MOVL C00363 V=800.0 PL=0
MOVL C00364 V=800.0 PL=0
MOVL C00365 V=800.0 PL=0
MOVL C00366 V=800.0 PL=0
MOVL C00367 V=800.0 PL=0
MOVL C00368 V=800.0 PL=0
MOVL C00369 V=800.0 PL=0
MOVL C00370 V=800.0 PL=0
MOVL C00371 V=800.0 PL=0
MOVL C00372 V=800.0 PL=0
MOVL C00373 V=800.0 PL=0
MOVL C00374 V=800.0 PL=0
MOVL C00375 V=800.0 PL=0
MOVL C00376 V=800.0 PL=0
MOVL C00377 V=800.0 PL=0
MOVL C00378 V=800.0 PL=0
MOVL C00379 V=800.0 PL=0
MOVL C00380 V=800.0 PL=0
MOVL C00381 V=800.0 PL=0
MOVL C00382 V=800.0 PL=0
MOVL C00383 V=800.0 PL=0
MOVL C00384 V=800.0 PL=0
MOVL C00385 V=800.0 PL=0
MOVL C00386 V=800.0 PL=0
MOVL C00387 V=800.0 PL=0
MOVL C00388 V=800.0 PL=0
MOVL C00389 V=800.0 PL=0
MOVL C00390 V=800.0 PL=0
MOVL C00391 V=800.0 PL=0
MOVL C00392 V=800.0 PL=0
MOVL C00393 V=800.0 PL=0
MOVL C00394 V=800.0 PL=0
MOVL C00395 V=800.0 PL=0
MOVL C00396 V=800.0 PL=0
MOVL C00397 V=800.0 PL=0
MOVL C00398 V=800.0 PL=0
MOVL C00399 V=800.0 PL=0
MOVL C00400 V=800.0 PL=0
MOVL C00401 V=800.0 PL=0
MOVL C00402 V=800.0 PL=0
MOVL C00403 V=800.0 PL=0
MOVL C00404 V=800.0 PL=0
MOVL C00405 V=800.0 PL=0
MOVL C00406 V=800.0 PL=0
MOVL C00407 V=800.0 PL=0
MOVL C00408 V=800.0 PL=0
MOVL C00409 V=800.0 PL=0
MOVL C00410 V=800.0 PL=0
MOVL C00411 V=800.0 PL=0
MOVL C00412 V=800.0 PL=0
MOVL C00413 V=800.0 PL=0
MOVL C00414 V=800.0 PL=0
MOVL C00415 V=800.0 PL=0
MOVL C00416 V=800.0 PL=0
MOVL C00417 V=800.0 PL=0
MOVL C00418 V=800.0 PL=0
MOVL C00419 V=800.0 PL=0
MOVL C00420 V=800.0 PL=0
MOVL C00421 V=800.0 PL=0
MOVL C00422 V=800.0 PL=0
MOVL C00423 V=800.0 PL=0
MOVL C00424 V=800.0 PL=0
MOVL C00425 V=800.0 PL=0
MOVL C00426 V=800.0 PL=0
MOVL C00427 V=800.0 PL=0
MOVL C00428 V=800.0 PL=0
MOVL C00429 V=800.0 PL=0
MOVL C00430 V=800.0 PL=0
MOVL C00431 V=800.0 PL=0
MOVL C00432 V=800.0 PL=0
MOVL C00433 V=800.0 PL=0
MOVL C00434 V=800.0 PL=0
MOVL C00435 V=800.0 PL=0
MOVL C00436 V=800.0 PL=0
MOVL C00437 V=800.0 PL=0
MOVL C00438 V=800.0 PL=0
MOVL C00439 V=800.0 PL=0
MOVL C00440 V=800.0 PL=0
MOVL C00441 V=800.0 PL=0
MOVL C00442 V=800.0 PL=0
MOVL C00443 V=800.0 PL=0
MOVL C00444 V=800.0 PL=0
MOVL C00445 V=800.0 PL=0
MOVL C00446 V=800.0 PL=0
MOVL C00447 V=800.0 PL=0
MOVL C00448 V=800.0 PL=0
MOVL C00449 V=800.0 PL=0
MOVL C00450 V=800.0 PL=0
MOVL C00451 V=800.0 PL=0
MOVL C00452 V=800.0 PL=0
MOVL C00453 V=800.0 PL=0
MOVL C00454 V=800.0 PL=0
MOVL C00455 V=800.0 PL=0
MOVL C00456 V=800.0 PL=0
MOVL C00457 V=800.0 PL=0
MOVL C00458 V=800.0 PL=0
MOVL C00459 V=800.0 PL=0
MOVL C00460 V=800.0 PL=0
MOVL C00461 V=800.0 PL=0
MOVL C00462 V=800.0 PL=0
MOVL C00463 V=800.0 PL=0
MOVL C00464 V=800.0 PL=0
MOVL C00465 V=800.0 PL=0
MOVL C00466 V=800.0 PL=0
MOVL C00467 V=800.0 PL=0
MOVL C00468 V=800.0 PL=0
MOVL C00469 V=800.0 PL=0
MOVL C00470 V=800.0 PL=0
MOVL C00471 V=800.0 PL=0
MOVL C00472 V=800.0 PL=0
MOVL C00473 V=800.0 PL=0
MOVL C00474 V=800.0 PL=0
MOVL C00475 V=800.0 PL=0
MOVL C00476 V=800.0 PL=0
MOVL C00477 V=800.0 PL=0
MOVL C00478 V=800.0 PL=0
MOVL C00479 V=800.0 PL=0
MOVL C00480 V=800.0 PL=0
MOVL C00481 V=800.0 PL=0
MOVL C00482 V=800.0 PL=0
MOVL C00483 V=800.0 PL=0
MOVL C00484 V=800.0 PL=0
MOVL C00485 V=800.0 PL=0
MOVL C00486 V=800.0 PL=0
MOVL C00487 V=800.0 PL=0
MOVL C00488 V=800.0 PL=0
MOVL C00489 V=800.0 PL=0
MOVL C00490 V=800.0 PL=0
MOVL C00491 V=800.0 PL=0
MOVL C00492 V=800.0 PL=0
MOVL C00493 V=800.0 PL=0
MOVL C00494 V=800.0 PL=0
MOVL C00495 V=800.0 PL=0
MOVL C00496 V=800.0 PL=0
MOVL C00497 V=800.0 PL=0
MOVL C00498 V=800.0 PL=0
MOVL C00499 V=800.0 PL=0
MOVL C00500 V=800.0 PL=0
MOVL C00501 V=800.0 PL=0
MOVL C00502 V=800.0 PL=0
MOVL C00503 V=800.0 PL=0
MOVL C00504 V=800.0 PL=0
MOVL C00505 V=800.0 PL=0
MOVL C00506 V=800.0 PL=0
MOVL C00507 V=800.0 PL=0
MOVL C00508 V=800.0 PL=0
MOVL C00509 V=800.0 PL=0
MOVL C00510 V=800.0 PL=0
MOVL C00511 V=800.0 PL=0
MOVL C00512 V=800.0 PL=0
MOVL C00513 V=800.0 PL=0
MOVL C00514 V=800.0 PL=0
MOVL C00515 V=800.0 PL=0
MOVL C00516 V=800.0 PL=0
MOVL C00517 V=800.0 PL=0
MOVL C00518 V=800.0 PL=0
MOVL C00519 V=800.0 PL=0
MOVL C00520 V=800.0 PL=0
MOVL C00521 V=800.0 PL=0
MOVL C00522 V=800.0 PL=0
MOVL C00523 V=800.0 PL=0
MOVL C00524 V=800.0 PL=0
MOVL C00525 V=800.0 PL=0
MOVL C00526 V=800.0 PL=0
MOVL C00527 V=800.0 PL=0
MOVL C00528 V=800.0 PL=0
MOVL C00529 V=800.0 PL=0
MOVL C00530 V=800.0 PL=0
MOVL C00531 V=800.0 PL=0
MOVL C00532 V=800.0 PL=0
MOVL C00533 V=800.0 PL=0
MOVL C00534 V=800.0 PL=0
MOVL C00535 V=800.0 PL=0
MOVL C00536 V=800.0 PL=0
MOVL C00537 V=800.0 PL=0
MOVL C00538 V=800.0 PL=0
MOVL C00539 V=800.0 PL=0
MOVL C00540 V=800.0 PL=0
MOVL C00541 V=800.0 PL=0
MOVL C00542 V=800.0 PL=0
MOVL C00543 V=800.0 PL=0
MOVL C00544 V=800.0 PL=0
MOVL C00545 V=800.0 PL=0
MOVL C00546 V=800.0 PL=0
MOVL C00547 V=800.0 PL=0
MOVL C00548 V=800.0 PL=0
MOVL C00549 V=800.0 PL=0
MOVL C00550 V=800.0 PL=0
MOVL C00551 V=800.0 PL=0
MOVL C00552 V=800.0 PL=0
MOVL C00553 V=800.0 PL=0
MOVL C00554 V=800.0 PL=0
MOVL C00555 V=800.0 PL=0
MOVL C00556 V=800.0 PL=0
MOVL C00557 V=800.0 PL=0
MOVL C00558 V=800.0 PL=0
MOVL C00559 V=800.0 PL=0
MOVL C00560 V=800.0 PL=0
MOVL C00561 V=800.0 PL=0
MOVL C00562 V=800.0 PL=0
MOVL C00563 V=800.0 PL=0
MOVL C00564 V=800.0 PL=0
MOVL C00565 V=800.0 PL=0
MOVL C00566 V=800.0 PL=0
MOVL C00567 V=800.0 PL=0
MOVL C00568 V=800.0 PL=0
MOVL C00569 V=800.0 PL=0
MOVL C00570 V=800.0 PL=0
MOVL C00571 V=800.0 PL=0
MOVL C00572 V=800.0 PL=0
MOVL C00573 V=800.0 PL=0
MOVL C00574 V=800.0 PL=0
MOVL C00575 V=800.0 PL=0
MOVL C00576 V=800.0 PL=0
MOVL C00577 V=800.0 PL=0
MOVL C00578 V=800.0 PL=0
MOVL C00579 V=800.0 PL=0
MOVL C00580 V=800.0 PL=0
MOVL C00581 V=800.0 PL=0
MOVL C00582 V=800.0 PL=0
MOVL C00583 V=800.0 PL=0
MOVL C00584 V=800.0 PL=0
MOVL C00585 V=800.0 PL=0
MOVL C00586 V=800.0 PL=0
MOVL C00587 V=800.0 PL=0
MOVL C00588 V=800.0 PL=0
MOVL C00589 V=800.0 PL=0
MOVL C00590 V=800.0 PL=0
MOVL C00591 V=800.0 PL=0
MOVL C00592 V=800.0 PL=0
MOVL C00593 V=800.0 PL=0
MOVL C00594 V=800.0 PL=0
MOVL C00595 V=800.0 PL=0
MOVL C00596 V=800.0 PL=0
MOVL C00597 V=800.0 PL=0
MOVL C00598 V=800.0 PL=0
MOVL C00599 V=800.0 PL=0
MOVL C00600 V=800.0 PL=0
MOVL C00601 V=800.0 PL=0
MOVL C00602 V=800.0 PL=0
MOVL C00603 V=800.0 PL=0
MOVL C00604 V=800.0 PL=0
MOVL C00605 V=800.0 PL=0
MOVL C00606 V=800.0 PL=0
MOVL C00607 V=800.0 PL=0
MOVL C00608 V=800.0 PL=0
MOVL C00609 V=800.0 PL=0
MOVL C00610 V=800.0 PL=0
MOVL C00611 V=800.0 PL=0
MOVL C00612 V=800.0 PL=0
MOVL C00613 V=800.0 PL=0
MOVL C00614 V=800.0 PL=0
MOVL C00615 V=800.0 PL=0
MOVL C00616 V=800.0 PL=0
MOVL C00617 V=800.0 PL=0
MOVL C00618 V=800.0 PL=0
MOVL C00619 V=800.0 PL=0
MOVL C00620 V=800.0 PL=0
MOVL C00621 V=800.0 PL=0
MOVL C00622 V=800.0 PL=0
MOVL C00623 V=800.0 PL=0
MOVL C00624 V=800.0 PL=0
MOVL C00625 V=800.0 PL=0
MOVL C00626 V=800.0 PL=0
MOVL C00627 V=800.0 PL=0
MOVL C00628 V=800.0 PL=0
MOVL C00629 V=800.0 PL=0
MOVL C00630 V=800.0 PL=0
MOVL C00631 V=800.0 PL=0
MOVL C00632 V=800.0 PL=0
MOVL C00633 V=800.0 PL=0
MOVL C00634 V=800.0 PL=0
MOVL C00635 V=800.0 PL=0
MOVL C00636 V=800.0 PL=0
MOVL C00637 V=800.0 PL=0
MOVL C00638 V=800.0 PL=0
MOVL C00639 V=800.0 PL=0
MOVL C00640 V=800.0 PL=0
MOVL C00641 V=800.0 PL=0
MOVL C00642 V=800.0 PL=0
MOVL C00643 V=800.0 PL=0
MOVL C00644 V=800.0 PL=0
MOVL C00645 V=800.0 PL=0
MOVL C00646 V=800.0 PL=0
MOVL C00647 V=800.0 PL=0
MOVL C00648 V=800.0 PL=0
MOVL C00649 V=800.0 PL=0
MOVL C00650 V=800.0 PL=0
MOVL C00651 V=800.0 PL=0
MOVL C00652 V=800.0 PL=0
MOVL C00653 V=800.0 PL=0
MOVL C00654 V=800.0 PL=0
MOVL C00655 V=800.0 PL=0
MOVL C00656 V=800.0 PL=0
MOVL C00657 V=800.0 PL=0
MOVL C00658 V=800.0 PL=0
MOVL C00659 V=800.0 PL=0
MOVL C00660 V=800.0 PL=0
MOVL C00661 V=800.0 PL=0
MOVL C00662 V=800.0 PL=0
MOVL C00663 V=800.0 PL=0
MOVL C00664 V=800.0 PL=0
MOVL C00665 V=800.0 PL=0
MOVL C00666 V=800.0 PL=0
MOVL C00667 V=800.0 PL=0
MOVL C00668 V=800.0 PL=0
MOVL C00669 V=800.0 PL=0
MOVL C00670 V=800.0 PL=0
MOVL C00671 V=800.0 PL=0
MOVL C00672 V=800.0 PL=0
MOVL C00673 V=800.0 PL=0
MOVL C00674 V=800.0 PL=0
MOVL C00675 V=800.0 PL=0
MOVL C00676 V=800.0 PL=0
MOVL C00677 V=800.0 PL=0
MOVL C00678 V=800.0 PL=0
MOVL C00679 V=800.0 PL=0
MOVL C00680 V=800.0 PL=0
MOVL C00681 V=800.0 PL=0
MOVL C00682 V=800.0 PL=0
MOVL C00683 V=800.0 PL=0
MOVL C00684 V=800.0 PL=0
MOVL C00685 V=800.0 PL=0
MOVL C00686 V=800.0 PL=0
MOVL C00687 V=800.0 PL=0
MOVL C00688 V=800.0 PL=0
MOVL C00689 V=800.0 PL=0
MOVL C00690 V=800.0 PL=0
MOVL C00691 V=800.0 PL=0
MOVL C00692 V=800.0 PL=0
MOVL C00693 V=800.0 PL=0
MOVL C00694 V=800.0 PL=0
MOVL C00695 V=800.0 PL=0
MOVL C00696 V=800.0 PL=0
MOVL C00697 V=800.0 PL=0
MOVL C00698 V=800.0 PL=0
MOVL C00699 V=800.0 PL=0
MOVL C00700 V=800.0 PL=0
MOVL C00701 V=800.0 PL=0
MOVL C00702 V=800.0 PL=0
MOVL C00703 V=800.0 PL=0
MOVL C00704 V=800.0 PL=0
MOVL C00705 V=800.0 PL=0
MOVL C00706 V=800.0 PL=0
MOVL C00707 V=800.0 PL=0
MOVL C00708 V=800.0 PL=0
MOVL C00709 V=800.0 PL=0
MOVL C00710 V=800.0 PL=0
MOVL C00711 V=800.0 PL=0
MOVL C00712 V=800.0 PL=0
MOVL C00713 V=800.0 PL=0
MOVL C00714 V=800.0 PL=0
MOVL C00715 V=800.0 PL=0
MOVL C00716 V=800.0 PL=0
MOVL C00717 V=800.0 PL=0
MOVL C00718 V=800.0 PL=0
MOVL C00719 V=800.0 PL=0
MOVL C00720 V=800.0 PL=0
MOVL C00721 V=800.0 PL=0
MOVL C00722 V=800.0 PL=0
MOVL C00723 V=800.0 PL=0
MOVL C00724 V=800.0 PL=0
MOVL C00725 V=800.0 PL=0
MOVL C00726 V=800.0 PL=0
MOVL C00727 V=800.0 PL=0
MOVL C00728 V=800.0 PL=0
MOVL C00729 V=800.0 PL=0
MOVL C00730 V=800.0 PL=0
MOVL C00731 V=800.0 PL=0
MOVL C00732 V=800.0 PL=0
MOVL C00733 V=800.0 PL=0
MOVL C00734 V=800.0 PL=0
MOVL C00735 V=800.0 PL=0
MOVL C00736 V=800.0 PL=0
MOVL C00737 V=800.0 PL=0
MOVL C00738 V=800.0 PL=0
MOVL C00739 V=800.0 PL=0
MOVL C00740 V=800.0 PL=0
MOVL C00741 V=800.0 PL=0
MOVL C00742 V=800.0 PL=0
MOVL C00743 V=800.0 PL=0
MOVL C00744 V=800.0 PL=0
MOVL C00745 V=800.0 PL=0
MOVL C00746 V=800.0 PL=0
MOVL C00747 V=800.0 PL=0
MOVL C00748 V=800.0 PL=0
MOVL C00749 V=800.0 PL=0
MOVL C00750 V=800.0 PL=0
MOVL C00751 V=800.0 PL=0
MOVL C00752 V=800.0 PL=0
MOVL C00753 V=800.0 PL=0
MOVL C00754 V=800.0 PL=0
MOVL C00755 V=800.0 PL=0
MOVL C00756 V=800.0 PL=0
MOVL C00757 V=800.0 PL=0
MOVL C00758 V=800.0 PL=0
MOVL C00759 V=800.0 PL=0
MOVL C00760 V=800.0 PL=0
MOVL C00761 V=800.0 PL=0
MOVL C00762 V=800.0 PL=0
MOVL C00763 V=800.0 PL=0
MOVL C00764 V=800.0 PL=0
MOVL C00765 V=800.0 PL=0
MOVL C00766 V=800.0 PL=0
MOVL C00767 V=800.0 PL=0
MOVL C00768 V=800.0 PL=0
MOVL C00769 V=800.0 PL=0
MOVL C00770 V=800.0 PL=0
MOVL C00771 V=800.0 PL=0
MOVL C00772 V=800.0 PL=0
MOVL C00773 V=800.0 PL=0
MOVL C00774 V=800.0 PL=0
MOVL C00775 V=800.0 PL=0
MOVL C00776 V=800.0 PL=0
MOVL C00777 V=800.0 PL=0
MOVL C00778 V=800.0 PL=0
MOVL C00779 V=800.0 PL=0
MOVL C00780 V=800.0 PL=0
MOVL C00781 V=800.0 PL=0
MOVL C00782 V=800.0 PL=0
MOVL C00783 V=800.0 PL=0
MOVL C00784 V=800.0 PL=0
MOVL C00785 V=800.0 PL=0
MOVL C00786 V=800.0 PL=0
MOVL C00787 V=800.0 PL=0
MOVL C00788 V=800.0 PL=0
MOVL C00789 V=800.0 PL=0
MOVL C00790 V=800.0 PL=0
MOVL C00791 V=800.0 PL=0
MOVL C00792 V=800.0 PL=0
MOVL C00793 V=800.0 PL=0
MOVL C00794 V=800.0 PL=0
MOVL C00795 V=800.0 PL=0
MOVL C00796 V=800.0 PL=0
MOVL C00797 V=800.0 PL=0
MOVL C00798 V=800.0 PL=0
MOVL C00799 V=800.0 PL=0
MOVL C00800 V=800.0 PL=0
MOVL C00801 V=800.0 PL=0
MOVL C00802 V=800.0 PL=0
MOVL C00803 V=800.0 PL=0
MOVL C00804 V=800.0 PL=0
MOVL C00805 V=800.0 PL=0
MOVL C00806 V=800.0 PL=0
MOVL C00807 V=800.0 PL=0
MOVL C00808 V=800.0 PL=0
MOVL C00809 V=800.0 PL=0
MOVL C00810 V=800.0 PL=0
MOVL C00811 V=800.0 PL=0
MOVL C00812 V=800.0 PL=0
MOVL C00813 V=800.0 PL=0
MOVL C00814 V=800.0 PL=0
MOVL C00815 V=800.0 PL=0
MOVL C00816 V=800.0 PL=0
MOVL C00817 V=800.0 PL=0
MOVL C00818 V=800.0 PL=0
MOVL C00819 V=800.0 PL=0
MOVL C00820 V=800.0 PL=0
MOVL C00821 V=800.0 PL=0
MOVL C00822 V=800.0 PL=0
MOVL C00823 V=800.0 PL=0
MOVL C00824 V=800.0 PL=0
MOVL C00825 V=800.0 PL=0
MOVL C00826 V=800.0 PL=0
MOVL C00827 V=800.0 PL=0
MOVL C00828 V=800.0 PL=0
MOVL C00829 V=800.0 PL=0
MOVL C00830 V=800.0 PL=0
MOVL C00831 V=800.0 PL=0
MOVL C00832 V=800.0 PL=0
MOVL C00833 V=800.0 PL=0
MOVL C00834 V=800.0 PL=0
MOVL C00835 V=800.0 PL=0
MOVL C00836 V=800.0 PL=0
MOVL C00837 V=800.0 PL=0
MOVL C00838 V=800.0 PL=0
MOVL C00839 V=800.0 PL=0
MOVL C00840 V=800.0 PL=0
MOVL C00841 V=800.0 PL=0
MOVL C00842 V=800.0 PL=0
MOVL C00843 V=800.0 PL=0
MOVL C00844 V=800.0 PL=0
MOVL C00845 V=800.0 PL=0
MOVL C00846 V=800.0 PL=0
MOVL C00847 V=800.0 PL=0
MOVL C00848 V=800.0 PL=0
MOVL C00849 V=800.0 PL=0
MOVL C00850 V=800.0 PL=0
MOVL C00851 V=800.0 PL=0
MOVL C00852 V=800.0 PL=0
MOVL C00853 V=800.0 PL=0
MOVL C00854 V=800.0 PL=0
MOVL C00855 V=800.0 PL=0
MOVL C00856 V=800.0 PL=0
MOVL C00857 V=800.0 PL=0
MOVL C00858 V=800.0 PL=0
MOVL C00859 V=800.0 PL=0
MOVL C00860 V=800.0 PL=0
MOVL C00861 V=800.0 PL=0
MOVL C00862 V=800.0 PL=0
MOVL C00863 V=800.0 PL=0
MOVL C00864 V=800.0 PL=0
MOVL C00865 V=800.0 PL=0
MOVL C00866 V=800.0 PL=0
MOVL C00867 V=800.0 PL=0
MOVL C00868 V=800.0 PL=0
MOVL C00869 V=800.0 PL=0
MOVL C00870 V=800.0 PL=0
MOVL C00871 V=800.0 PL=0
MOVL C00872 V=800.0 PL=0
MOVL C00873 V=800.0 PL=0
MOVL C00874 V=800.0 PL=0
MOVL C00875 V=800.0 PL=0
MOVL C00876 V=800.0 PL=0
MOVL C00877 V=800.0 PL=0
MOVL C00878 V=800.0 PL=0
MOVL C00879 V=800.0 PL=0
MOVL C00880 V=800.0 PL=0
MOVL C00881 V=800.0 PL=0
MOVL C00882 V=800.0 PL=0
MOVL C00883 V=800.0 PL=0
MOVL C00884 V=800.0 PL=0
MOVL C00885 V=800.0 PL=0
MOVL C00886 V=800.0 PL=0
MOVL C00887 V=800.0 PL=0
MOVL C00888 V=800.0 PL=0
MOVL C00889 V=800.0 PL=0
MOVL C00890 V=800.0 PL=0
MOVL C00891 V=800.0 PL=0
MOVL C00892 V=800.0 PL=0
MOVL C00893 V=800.0 PL=0
MOVL C00894 V=800.0 PL=0
MOVL C00895 V=800.0 PL=0
MOVL C00896 V=800.0 PL=0
MOVL C00897 V=800.0 PL=0
MOVL C00898 V=800.0 PL=0
MOVL C00899 V=800.0 PL=0
MOVL C00900 V=800.0 PL=0
MOVL C00901 V=800.0 PL=0
MOVL C00902 V=800.0 PL=0
MOVL C00903 V=800.0 PL=0
MOVL C00904 V=800.0 PL=0
MOVL C00905 V=800.0 PL=0
MOVL C00906 V=800.0 PL=0
MOVL C00907 V=800.0 PL=0
MOVL C00908 V=800.0 PL=0
MOVL C00909 V=800.0 PL=0
MOVL C00910 V=800.0 PL=0
MOVL C00911 V=800.0 PL=0
MOVL C00912 V=800.0 PL=0
MOVL C00913 V=800.0 PL=0
MOVL C00914 V=800.0 PL=0
MOVL C00915 V=800.0 PL=0
MOVL C00916 V=800.0 PL=0
MOVL C00917 V=800.0 PL=0
MOVL C00918 V=800.0 PL=0
MOVL C00919 V=800.0 PL=0
MOVL C00920 V=800.0 PL=0
MOVL C00921 V=800.0 PL=0
MOVL C00922 V=800.0 PL=0
MOVL C00923 V=800.0 PL=0
MOVL C00924 V=800.0 PL=0
MOVL C00925 V=800.0 PL=0
MOVL C00926 V=800.0 PL=0
MOVL C00927 V=800.0 PL=0
MOVL C00928 V=800.0 PL=0
MOVL C00929 V=800.0 PL=0
MOVL C00930 V=800.0 PL=0
MOVL C00931 V=800.0 PL=0
MOVL C00932 V=800.0 PL=0
MOVL C00933 V=800.0 PL=0
MOVL C00934 V=800.0 PL=0
MOVL C00935 V=800.0 PL=0
MOVL C00936 V=800.0 PL=0
MOVL C00937 V=800.0 PL=0
MOVL C00938 V=800.0 PL=0
MOVL C00939 V=800.0 PL=0
MOVL C00940 V=800.0 PL=0
MOVL C00941 V=800.0 PL=0
MOVL C00942 V=800.0 PL=0
MOVL C00943 V=800.0 PL=0
MOVL C00944 V=800.0 PL=0
MOVL C00945 V=800.0 PL=0
MOVL C00946 V=800.0 PL=0
MOVL C00947 V=800.0 PL=0
MOVL C00948 V=800.0 PL=0
MOVL C00949 V=800.0 PL=0
MOVL C00950 V=800.0 PL=0
MOVL C00951 V=800.0 PL=0
MOVL C00952 V=800.0 PL=0
MOVL C00953 V=800.0 PL=0
MOVL C00954 V=800.0 PL=0
MOVL C00955 V=800.0 PL=0
MOVL C00956 V=800.0 PL=0
MOVL C00957 V=800.0 PL=0
MOVL C00958 V=800.0 PL=0
MOVL C00959 V=800.0 PL=0
MOVL C00960 V=800.0 PL=0
MOVL C00961 V=800.0 PL=0
MOVL C00962 V=800.0 PL=0
MOVL C00963 V=800.0 PL=0
MOVL C00964 V=800.0 PL=0
MOVL C00965 V=800.0 PL=0
MOVL C00966 V=800.0 PL=0
MOVL C00967 V=800.0 PL=0
MOVL C00968 V=800.0 PL=0
MOVL C00969 V=800.0 PL=0
MOVL C00970 V=800.0 PL=0
MOVL C00971 V=800.0 PL=0
MOVL C00972 V=800.0 PL=0
MOVL C00973 V=800.0 PL=0
MOVL C00974 V=800.0 PL=0
MOVL C00975 V=800.0 PL=0
MOVL C00976 V=800.0 PL=0
MOVL C00977 V=800.0 PL=0
MOVL C00978 V=800.0 PL=0
MOVL C00979 V=800.0 PL=0
MOVL C00980 V=800.0 PL=0
MOVL C00981 V=800.0 PL=0
MOVL C00982 V=800.0 PL=0
MOVL C00983 V=800.0 PL=0
MOVL C00984 V=800.0 PL=0
MOVL C00985 V=800.0 PL=0
MOVL C00986 V=800.0 PL=0
MOVL C00987 V=800.0 PL=0
MOVL C00988 V=800.0 PL=0
MOVL C00989 V=800.0 PL=0
MOVL C00990 V=800.0 PL=0
MOVL C00991 V=800.0 PL=0
MOVL C00992 V=800.0 PL=0
MOVL C00993 V=800.0 PL=0
MOVL C00994 V=800.0 PL=0
MOVL C00995 V=800.0 PL=0
MOVL C00996 V=800.0 PL=0
MOVL C00997 V=800.0 PL=0
MOVL C00998 V=800.0 PL=0
MOVL C00999 V=800.0 PL=0
MOVL C01000 V=800.0 PL=0
MOVL C01001 V=800.0 PL=0
MOVL C01002 V=800.0 PL=0
MOVL C01003 V=800.0 PL=0
MOVL C01004 V=800.0 PL=0
MOVL C01005 V=800.0 PL=0
MOVL C01006 V=800.0 PL=0
MOVL C01007 V=800.0 PL=0
MOVL C01008 V=800.0 PL=0
MOVL C01009 V=800.0 PL=0
MOVL C01010 V=800.0 PL=0
MOVL C01011 V=800.0 PL=0
MOVL C01012 V=800.0 PL=0
MOVL C01013 V=800.0 PL=0
MOVL C01014 V=800.0 PL=0
MOVL C01015 V=800.0 PL=0
MOVL C01016 V=800.0 PL=0
MOVL C01017 V=800.0 PL=0
MOVL C01018 V=800.0 PL=0
MOVL C01019 V=800.0 PL=0
MOVL C01020 V=800.0 PL=0
MOVL C01021 V=800.0 PL=0
MOVL C01022 V=800.0 PL=0
MOVL C01023 V=800.0 PL=0
MOVL C01024 V=800.0 PL=0
MOVL C01025 V=800.0 PL=0
MOVL C01026 V=800.0 PL=0
MOVL C01027 V=800.0 PL=0
MOVL C01028 V=800.0 PL=0
MOVL C01029 V=800.0 PL=0
MOVL C01030 V=800.0 PL=0
MOVL C01031 V=800.0 PL=0
MOVL C01032 V=800.0 PL=0
MOVL C01033 V=800.0 PL=0
MOVL C01034 V=800.0 PL=0
MOVL C01035 V=800.0 PL=0
MOVL C01036 V=800.0 PL=0
MOVL C01037 V=800.0 PL=0
MOVL C01038 V=800.0 PL=0
MOVL C01039 V=800.0 PL=0
MOVL C01040 V=800.0 PL=0
MOVL C01041 V=800.0 PL=0
MOVL C01042 V=800.0 PL=0
MOVL C01043 V=800.0 PL=0
MOVL C01044 V=800.0 PL=0
MOVL C01045 V=800.0 PL=0
MOVL C01046 V=800.0 PL=0
MOVL C01047 V=800.0 PL=0
MOVL C01048 V=800.0 PL=0
MOVL C01049 V=800.0 PL=0
MOVL C01050 V=800.0 PL=0
MOVL C01051 V=800.0 PL=0
MOVL C01052 V=800.0 PL=0
MOVL C01053 V=800.0 PL=0
MOVL C01054 V=800.0 PL=0
MOVL C01055 V=800.0 PL=0
MOVL C01056 V=800.0 PL=0
MOVL C01057 V=800.0 PL=0
MOVL C01058 V=800.0 PL=0
MOVL C01059 V=800.0 PL=0
MOVL C01060 V=800.0 PL=0
MOVL C01061 V=800.0 PL=0
MOVL C01062 V=800.0 PL=0
MOVL C01063 V=800.0 PL=0
MOVL C01064 V=800.0 PL=0
MOVL C01065 V=800.0 PL=0
MOVL C01066 V=800.0 PL=0
MOVL C01067 V=800.0 PL=0
MOVL C01068 V=800.0 PL=0
MOVL C01069 V=800.0 PL=0
MOVL C01070 V=800.0 PL=0
MOVL C01071 V=800.0 PL=0
MOVL C01072 V=800.0 PL=0
MOVL C01073 V=800.0 PL=0
MOVL C01074 V=800.0 PL=0
MOVL C01075 V=800.0 PL=0
MOVL C01076 V=800.0 PL=0
MOVL C01077 V=800.0 PL=0
MOVL C01078 V=800.0 PL=0
MOVL C01079 V=800.0 PL=0
MOVL C01080 V=800.0 PL=0
MOVL C01081 V=800.0 PL=0
MOVL C01082 V=800.0 PL=0
MOVL C01083 V=800.0 PL=0
MOVL C01084 V=800.0 PL=0
MOVL C01085 V=800.0 PL=0
MOVL C01086 V=800.0 PL=0
MOVL C01087 V=800.0 PL=0
MOVL C01088 V=800.0 PL=0
MOVL C01089 V=800.0 PL=0
MOVL C01090 V=800.0 PL=0
MOVL C01091 V=800.0 PL=0
MOVL C01092 V=800.0 PL=0
MOVL C01093 V=800.0 PL=0
MOVL C01094 V=800.0 PL=0
MOVL C01095 V=800.0 PL=0
MOVL C01096 V=800.0 PL=0
MOVL C01097 V=800.0 PL=0
MOVL C01098 V=800.0 PL=0
MOVL C01099 V=800.0 PL=0
MOVL C01100 V=800.0 PL=0
MOVL C01101 V=800.0 PL=0
MOVL C01102 V=800.0 PL=0
MOVL C01103 V=800.0 PL=0
MOVL C01104 V=800.0 PL=0
MOVL C01105 V=800.0 PL=0
MOVL C01106 V=800.0 PL=0
MOVL C01107 V=800.0 PL=0
MOVL C01108 V=800.0 PL=0
MOVL C01109 V=800.0 PL=0
MOVL C01110 V=800.0 PL=0
MOVL C01111 V=800.0 PL=0
MOVL C01112 V=800.0 PL=0
MOVL C01113 V=800.0 PL=0
MOVL C01114 V=800.0 PL=0
MOVL C01115 V=800.0 PL=0
MOVL C01116 V=800.0 PL=0
MOVL C01117 V=800.0 PL=0
MOVL C01118 V=800.0 PL=0
MOVL C01119 V=800.0 PL=0
MOVL C01120 V=800.0 PL=0
MOVL C01121 V=800.0 PL=0
MOVL C01122 V=800.0 PL=0
MOVL C01123 V=800.0 PL=0
MOVL C01124 V=800.0 PL=0
MOVL C01125 V=800.0 PL=0
MOVL C01126 V=800.0 PL=0
MOVL C01127 V=800.0 PL=0
MOVL C01128 V=800.0 PL=0
MOVL C01129 V=800.0 PL=0
MOVL C01130 V=800.0 PL=0
MOVL C01131 V=800.0 PL=0
MOVL C01132 V=800.0 PL=0
MOVL C01133 V=800.0 PL=0
MOVL C01134 V=800.0 PL=0
MOVL C01135 V=800.0 PL=0
MOVL C01136 V=800.0 PL=0
MOVL C01137 V=800.0 PL=0
MOVL C01138 V=800.0 PL=0
MOVL C01139 V=800.0 PL=0
MOVL C01140 V=800.0 PL=0
MOVL C01141 V=800.0 PL=0
MOVL C01142 V=800.0 PL=0
MOVL C01143 V=800.0 PL=0
MOVL C01144 V=800.0 PL=0
MOVL C01145 V=800.0 PL=0
MOVL C01146 V=800.0 PL=0
MOVL C01147 V=800.0 PL=0
MOVL C01148 V=800.0 PL=0
MOVL C01149 V=800.0 PL=0
MOVL C01150 V=800.0 PL=0
MOVL C01151 V=800.0 PL=0
MOVL C01152 V=800.0 PL=0
MOVL C01153 V=800.0 PL=0
MOVL C01154 V=800.0 PL=0
MOVL C01155 V=800.0 PL=0
MOVL C01156 V=800.0 PL=0
MOVL C01157 V=800.0 PL=0
MOVL C01158 V=800.0 PL=0
MOVL C01159 V=800.0 PL=0
MOVL C01160 V=800.0 PL=0
MOVL C01161 V=800.0 PL=0
MOVL C01162 V=800.0 PL=0
MOVL C01163 V=800.0 PL=0
MOVL C01164 V=800.0 PL=0
MOVL C01165 V=800.0 PL=0
MOVL C01166 V=800.0 PL=0
MOVL C01167 V=800.0 PL=0
MOVL C01168 V=800.0 PL=0
MOVL C01169 V=800.0 PL=0
MOVL C01170 V=800.0 PL=0
MOVL C01171 V=800.0 PL=0
MOVL C01172 V=800.0 PL=0
MOVL C01173 V=800.0 PL=0
MOVL C01174 V=800.0 PL=0
MOVL C01175 V=800.0 PL=0
MOVL C01176 V=800.0 PL=0
MOVL C01177 V=800.0 PL=0
MOVL C01178 V=800.0 PL=0
MOVL C01179 V=800.0 PL=0
MOVL C01180 V=800.0 PL=0
MOVL C01181 V=800.0 PL=0
MOVL C01182 V=800.0 PL=0
MOVL C01183 V=800.0 PL=0
MOVL C01184 V=800.0 PL=0
MOVL C01185 V=800.0 PL=0
MOVL C01186 V=800.0 PL=0
MOVL C01187 V=800.0 PL=0
MOVL C01188 V=800.0 PL=0
MOVL C01189 V=800.0 PL=0
MOVL C01190 V=800.0 PL=0
MOVL C01191 V=800.0 PL=0
MOVL C01192 V=800.0 PL=0
MOVL C01193 V=800.0 PL=0
MOVL C01194 V=800.0 PL=0
MOVL C01195 V=800.0 PL=0
MOVL C01196 V=800.0 PL=0
MOVL C01197 V=800.0 PL=0
MOVL C01198 V=800.0 PL=0
MOVL C01199 V=800.0 PL=0
MOVL C01200 V=800.0 PL=0
MOVL C01201 V=800.0 PL=0
MOVL C01202 V=800.0 PL=0
MOVL C01203 V=800.0 PL=0
MOVL C01204 V=800.0 PL=0
MOVL C01205 V=800.0 PL=0
MOVL C01206 V=800.0 PL=0
MOVL C01207 V=800.0 PL=0
MOVL C01208 V=800.0 PL=0
MOVL C01209 V=800.0 PL=0
MOVL C01210 V=800.0 PL=0
MOVL C01211 V=800.0 PL=0
MOVL C01212 V=800.0 PL=0
MOVL C01213 V=800.0 PL=0
MOVL C01214 V=800.0 PL=0
MOVL C01215 V=800.0 PL=0
MOVL C01216 V=800.0 PL=0
MOVL C01217 V=800.0 PL=0
MOVL C01218 V=800.0 PL=0
MOVL C01219 V=800.0 PL=0
MOVL C01220 V=800.0 PL=0
MOVL C01221 V=800.0 PL=0
MOVL C01222 V=800.0 PL=0
MOVL C01223 V=800.0 PL=0
MOVL C01224 V=800.0 PL=0
MOVL C01225 V=800.0 PL=0
MOVL C01226 V=800.0 PL=0
MOVL C01227 V=800.0 PL=0
MOVL C01228 V=800.0 PL=0
MOVL C01229 V=800.0 PL=0
MOVL C01230 V=800.0 PL=0
MOVL C01231 V=800.0 PL=0
MOVL C01232 V=800.0 PL=0
MOVL C01233 V=800.0 PL=0
MOVL C01234 V=800.0 PL=0
MOVL C01235 V=800.0 PL=0
MOVL C01236 V=800.0 PL=0
MOVL C01237 V=800.0 PL=0
MOVL C01238 V=800.0 PL=0
MOVL C01239 V=800.0 PL=0
MOVL C01240 V=800.0 PL=0
MOVL C01241 V=800.0 PL=0
MOVL C01242 V=800.0 PL=0
MOVL C01243 V=800.0 PL=0
MOVL C01244 V=800.0 PL=0
MOVL C01245 V=800.0 PL=0
MOVL C01246 V=800.0 PL=0
MOVL C01247 V=800.0 PL=0
MOVL C01248 V=800.0 PL=0
MOVL C01249 V=800.0 PL=0
MOVL C01250 V=800.0 PL=0
MOVL C01251 V=800.0 PL=0
MOVL C01252 V=800.0 PL=0
MOVL C01253 V=800.0 PL=0
MOVL C01254 V=800.0 PL=0
MOVL C01255 V=800.0 PL=0
MOVL C01256 V=800.0 PL=0
MOVL C01257 V=800.0 PL=0
MOVL C01258 V=800.0 PL=0
MOVL C01259 V=800.0 PL=0
MOVL C01260 V=800.0 PL=0
MOVL C01261 V=800.0 PL=0
MOVL C01262 V=800.0 PL=0
MOVL C01263 V=800.0 PL=0
MOVL C01264 V=800.0 PL=0
MOVL C01265 V=800.0 PL=0
MOVL C01266 V=800.0 PL=0
MOVL C01267 V=800.0 PL=0
MOVL C01268 V=800.0 PL=0
MOVL C01269 V=800.0 PL=0
MOVL C01270 V=800.0 PL=0
MOVL C01271 V=800.0 PL=0
MOVL C01272 V=800.0 PL=0
MOVL C01273 V=800.0 PL=0
MOVL C01274 V=800.0 PL=0
MOVL C01275 V=800.0 PL=0
MOVL C01276 V=800.0 PL=0
MOVL C01277 V=800.0 PL=0
MOVL C01278 V=800.0 PL=0
MOVL C01279 V=800.0 PL=0
MOVL C01280 V=800.0 PL=0
MOVL C01281 V=800.0 PL=0
MOVL C01282 V=800.0 PL=0
MOVL C01283 V=800.0 PL=0
MOVL C01284 V=800.0 PL=0
MOVL C01285 V=800.0 PL=0
MOVL C01286 V=800.0 PL=0
MOVL C01287 V=800.0 PL=0
MOVL C01288 V=800.0 PL=0
MOVL C01289 V=800.0 PL=0
MOVL C01290 V=800.0 PL=0
MOVL C01291 V=800.0 PL=0
MOVL C01292 V=800.0 PL=0
MOVL C01293 V=800.0 PL=0
MOVL C01294 V=800.0 PL=0
MOVL C01295 V=800.0 PL=0
MOVL C01296 V=800.0 PL=0
MOVL C01297 V=800.0 PL=0
MOVL C01298 V=800.0 PL=0
MOVL C01299 V=800.0 PL=0
MOVL C01300 V=800.0 PL=0
MOVL C01301 V=800.0 PL=0
MOVL C01302 V=800.0 PL=0
MOVL C01303 V=800.0 PL=0
MOVL C01304 V=800.0 PL=0
MOVL C01305 V=800.0 PL=0
MOVL C01306 V=800.0 PL=0
MOVL C01307 V=800.0 PL=0
MOVL C01308 V=800.0 PL=0
MOVL C01309 V=800.0 PL=0
MOVL C01310 V=800.0 PL=0
MOVL C01311 V=800.0 PL=0
MOVL C01312 V=800.0 PL=0
MOVL C01313 V=800.0 PL=0
MOVL C01314 V=800.0 PL=0
MOVL C01315 V=800.0 PL=0
MOVL C01316 V=800.0 PL=0
MOVL C01317 V=800.0 PL=0
MOVL C01318 V=800.0 PL=0
MOVL C01319 V=800.0 PL=0
MOVL C01320 V=800.0 PL=0
MOVL C01321 V=800.0 PL=0
MOVL C01322 V=800.0 PL=0
MOVL C01323 V=800.0 PL=0
MOVL C01324 V=800.0 PL=0
MOVL C01325 V=800.0 PL=0
MOVL C01326 V=800.0 PL=0
MOVL C01327 V=800.0 PL=0
MOVL C01328 V=800.0 PL=0
MOVL C01329 V=800.0 PL=0
MOVL C01330 V=800.0 PL=0
MOVL C01331 V=800.0 PL=0
MOVL C01332 V=800.0 PL=0
MOVL C01333 V=800.0 PL=0
MOVL C01334 V=800.0 PL=0
MOVL C01335 V=800.0 PL=0
MOVL C01336 V=800.0 PL=0
MOVL C01337 V=800.0 PL=0
MOVL C01338 V=800.0 PL=0
MOVL C01339 V=800.0 PL=0
MOVL C01340 V=800.0 PL=0
MOVL C01341 V=800.0 PL=0
MOVL C01342 V=800.0 PL=0
MOVL C01343 V=800.0 PL=0
MOVL C01344 V=800.0 PL=0
MOVL C01345 V=800.0 PL=0
MOVL C01346 V=800.0 PL=0
MOVL C01347 V=800.0 PL=0
MOVL C01348 V=800.0 PL=0
MOVL C01349 V=800.0 PL=0
MOVL C01350 V=800.0 PL=0
MOVL C01351 V=800.0 PL=0
MOVL C01352 V=800.0 PL=0
MOVL C01353 V=800.0 PL=0
MOVL C01354 V=800.0 PL=0
MOVL C01355 V=800.0 PL=0
MOVL C01356 V=800.0 PL=0
MOVL C01357 V=800.0 PL=0
MOVL C01358 V=800.0 PL=0
MOVL C01359 V=800.0 PL=0
MOVL C01360 V=800.0 PL=0
MOVL C01361 V=800.0 PL=0
MOVL C01362 V=800.0 PL=0
MOVL C01363 V=800.0 PL=0
MOVL C01364 V=800.0 PL=0
MOVL C01365 V=800.0 PL=0
MOVL C01366 V=800.0 PL=0
MOVL C01367 V=800.0 PL=0
MOVL C01368 V=800.0 PL=0
MOVL C01369 V=800.0 PL=0
MOVL C01370 V=800.0 PL=0
MOVL C01371 V=800.0 PL=0
MOVL C01372 V=800.0 PL=0
MOVL C01373 V=800.0 PL=0
MOVL C01374 V=800.0 PL=0
MOVL C01375 V=800.0 PL=0
MOVL C01376 V=800.0 PL=0
MOVL C01377 V=800.0 PL=0
MOVL C01378 V=800.0 PL=0
MOVL C01379 V=800.0 PL=0
MOVL C01380 V=800.0 PL=0
MOVL C01381 V=800.0 PL=0
MOVL C01382 V=800.0 PL=0
MOVL C01383 V=800.0 PL=0
MOVL C01384 V=800.0 PL=0
MOVL C01385 V=800.0 PL=0
MOVL C01386 V=800.0 PL=0
MOVL C01387 V=800.0 PL=0
MOVL C01388 V=800.0 PL=0
MOVL C01389 V=800.0 PL=0
MOVL C01390 V=800.0 PL=0
MOVL C01391 V=800.0 PL=0
MOVL C01392 V=800.0 PL=0
MOVL C01393 V=800.0 PL=0
MOVL C01394 V=800.0 PL=0
MOVL C01395 V=800.0 PL=0
MOVL C01396 V=800.0 PL=0
MOVL C01397 V=800.0 PL=0
MOVL C01398 V=800.0 PL=0
MOVL C01399 V=800.0 PL=0
MOVL C01400 V=800.0 PL=0
MOVL C01401 V=800.0 PL=0
MOVL C01402 V=800.0 PL=0
MOVL C01403 V=800.0 PL=0
MOVL C01404 V=800.0 PL=0
MOVL C01405 V=800.0 PL=0
MOVL C01406 V=800.0 PL=0
MOVL C01407 V=800.0 PL=0
MOVL C01408 V=800.0 PL=0
MOVL C01409 V=800.0 PL=0
MOVL C01410 V=800.0 PL=0
MOVL C01411 V=800.0 PL=0
MOVL C01412 V=800.0 PL=0
MOVL C01413 V=800.0 PL=0
MOVL C01414 V=800.0 PL=0
MOVL C01415 V=800.0 PL=0
MOVL C01416 V=800.0 PL=0
MOVL C01417 V=800.0 PL=0
MOVL C01418 V=800.0 PL=0
MOVL C01419 V=800.0 PL=0
MOVL C01420 V=800.0 PL=0
MOVL C01421 V=800.0 PL=0
MOVL C01422 V=800.0 PL=0
MOVL C01423 V=800.0 PL=0
MOVL C01424 V=800.0 PL=0
MOVL C01425 V=800.0 PL=0
MOVL C01426 V=800.0 PL=0
MOVL C01427 V=800.0 PL=0
MOVL C01428 V=800.0 PL=0
MOVL C01429 V=800.0 PL=0
MOVL C01430 V=800.0 PL=0
MOVL C01431 V=800.0 PL=0
MOVL C01432 V=800.0 PL=0
MOVL C01433 V=800.0 PL=0
MOVL C01434 V=800.0 PL=0
MOVL C01435 V=800.0 PL=0
MOVL C01436 V=800.0 PL=0
MOVL C01437 V=800.0 PL=0
MOVL C01438 V=800.0 PL=0
MOVL C01439 V=800.0 PL=0
MOVL C01440 V=800.0 PL=0
MOVL C01441 V=800.0 PL=0
MOVL C01442 V=800.0 PL=0
MOVL C01443 V=800.0 PL=0
MOVL C01444 V=800.0 PL=0
MOVL C01445 V=800.0 PL=0
MOVL C01446 V=800.0 PL=0
MOVL C01447 V=800.0 PL=0
MOVL C01448 V=800.0 PL=0
MOVL C01449 V=800.0 PL=0
MOVL C01450 V=800.0 PL=0
MOVL C01451 V=800.0 PL=0
MOVL C01452 V=800.0 PL=0
MOVL C01453 V=800.0 PL=0
MOVL C01454 V=800.0 PL=0
MOVL C01455 V=800.0 PL=0
MOVL C01456 V=800.0 PL=0
MOVL C01457 V=800.0 PL=0
MOVL C01458 V=800.0 PL=0
MOVL C01459 V=800.0 PL=0
MOVL C01460 V=800.0 PL=0
MOVL C01461 V=800.0 PL=0
MOVL C01462 V=800.0 PL=0
MOVL C01463 V=800.0 PL=0
MOVL C01464 V=800.0 PL=0
MOVL C01465 V=800.0 PL=0
MOVL C01466 V=800.0 PL=0
MOVL C01467 V=800.0 PL=0
MOVL C01468 V=800.0 PL=0
MOVL C01469 V=800.0 PL=0
MOVL C01470 V=800.0 PL=0
MOVL C01471 V=800.0 PL=0
MOVL C01472 V=800.0 PL=0
MOVL C01473 V=800.0 PL=0
MOVL C01474 V=800.0 PL=0
MOVL C01475 V=800.0 PL=0
MOVL C01476 V=800.0 PL=0
MOVL C01477 V=800.0 PL=0
MOVL C01478 V=800.0 PL=0
MOVL C01479 V=800.0 PL=0
MOVL C01480 V=800.0 PL=0
MOVL C01481 V=800.0 PL=0
MOVL C01482 V=800.0 PL=0
MOVL C01483 V=800.0 PL=0
MOVL C01484 V=800.0 PL=0
MOVL C01485 V=800.0 PL=0
MOVL C01486 V=800.0 PL=0
MOVL C01487 V=800.0 PL=0
MOVL C01488 V=800.0 PL=0
MOVL C01489 V=800.0 PL=0
MOVL C01490 V=800.0 PL=0
MOVL C01491 V=800.0 PL=0
MOVL C01492 V=800.0 PL=0
MOVL C01493 V=800.0 PL=0
MOVL C01494 V=800.0 PL=0
MOVL C01495 V=800.0 PL=0
MOVL C01496 V=800.0 PL=0
MOVL C01497 V=800.0 PL=0
MOVL C01498 V=800.0 PL=0
MOVL C01499 V=800.0 PL=0
MOVL C01500 V=800.0 PL=0
MOVL C01501 V=800.0 PL=0
MOVL C01502 V=800.0 PL=0
MOVL C01503 V=800.0 PL=0
MOVL C01504 V=800.0 PL=0
MOVL C01505 V=800.0 PL=0
MOVL C01506 V=800.0 PL=0
MOVL C01507 V=800.0 PL=0
MOVL C01508 V=800.0 PL=0
MOVL C01509 V=800.0 PL=0
MOVL C01510 V=800.0 PL=0
MOVL C01511 V=800.0 PL=0
MOVL C01512 V=800.0 PL=0
MOVL C01513 V=800.0 PL=0
MOVL C01514 V=800.0 PL=0
MOVL C01515 V=800.0 PL=0
MOVL C01516 V=800.0 PL=0
MOVL C01517 V=800.0 PL=0
MOVL C01518 V=800.0 PL=0
MOVL C01519 V=800.0 PL=0
MOVL C01520 V=800.0 PL=0
MOVL C01521 V=800.0 PL=0
MOVL C01522 V=800.0 PL=0
MOVL C01523 V=800.0 PL=0
MOVL C01524 V=800.0 PL=0
MOVL C01525 V=800.0 PL=0
MOVL C01526 V=800.0 PL=0
MOVL C01527 V=800.0 PL=0
MOVL C01528 V=800.0 PL=0
MOVL C01529 V=800.0 PL=0
MOVL C01530 V=800.0 PL=0
MOVL C01531 V=800.0 PL=0
MOVL C01532 V=800.0 PL=0
MOVL C01533 V=800.0 PL=0
MOVL C01534 V=800.0 PL=0
MOVL C01535 V=800.0 PL=0
MOVL C01536 V=800.0 PL=0
MOVL C01537 V=800.0 PL=0
MOVL C01538 V=800.0 PL=0
MOVL C01539 V=800.0 PL=0
MOVL C01540 V=800.0 PL=0
MOVL C01541 V=800.0 PL=0
MOVL C01542 V=800.0 PL=0
MOVL C01543 V=800.0 PL=0
MOVL C01544 V=800.0 PL=0
MOVL C01545 V=800.0 PL=0
MOVL C01546 V=800.0 PL=0
MOVL C01547 V=800.0 PL=0
MOVL C01548 V=800.0 PL=0
MOVL C01549 V=800.0 PL=0
MOVL C01550 V=800.0 PL=0
MOVL C01551 V=800.0 PL=0
MOVL C01552 V=800.0 PL=0
MOVL C01553 V=800.0 PL=0
MOVL C01554 V=800.0 PL=0
MOVL C01555 V=800.0 PL=0
MOVL C01556 V=800.0 PL=0
MOVL C01557 V=800.0 PL=0
MOVL C01558 V=800.0 PL=0
MOVL C01559 V=800.0 PL=0
MOVL C01560 V=800.0 PL=0
MOVL C01561 V=800.0 PL=0
MOVL C01562 V=800.0 PL=0
MOVL C01563 V=800.0 PL=0
MOVL C01564 V=800.0 PL=0
MOVL C01565 V=800.0 PL=0
MOVL C01566 V=800.0 PL=0
MOVL C01567 V=800.0 PL=0
MOVL C01568 V=800.0 PL=0
MOVL C01569 V=800.0 PL=0
MOVL C01570 V=800.0 PL=0
MOVL C01571 V=800.0 PL=0
MOVL C01572 V=800.0 PL=0
MOVL C01573 V=800.0 PL=0
MOVL C01574 V=800.0 PL=0
MOVL C01575 V=800.0 PL=0
MOVL C01576 V=800.0 PL=0
MOVL C01577 V=800.0 PL=0
MOVL C01578 V=800.0 PL=0
MOVL C01579 V=800.0 PL=0
MOVL C01580 V=800.0 PL=0
MOVL C01581 V=800.0 PL=0
MOVL C01582 V=800.0 PL=0
MOVL C01583 V=800.0 PL=0
MOVL C01584 V=800.0 PL=0
MOVL C01585 V=800.0 PL=0
MOVL C01586 V=800.0 PL=0
MOVL C01587 V=800.0 PL=0
MOVL C01588 V=800.0 PL=0
MOVL C01589 V=800.0 PL=0
MOVL C01590 V=800.0 PL=0
MOVL C01591 V=800.0 PL=0
MOVL C01592 V=800.0 PL=0
MOVL C01593 V=800.0 PL=0
MOVL C01594 V=800.0 PL=0
MOVL C01595 V=800.0 PL=0
MOVL C01596 V=800.0 PL=0
MOVL C01597 V=800.0 PL=0
MOVL C01598 V=800.0 PL=0
MOVL C01599 V=800.0 PL=0
MOVL C01600 V=800.0 PL=0
MOVL C01601 V=800.0 PL=0
MOVL C01602 V=800.0 PL=0
MOVL C01603 V=800.0 PL=0
MOVL C01604 V=800.0 PL=0
MOVL C01605 V=800.0 PL=0
MOVL C01606 V=800.0 PL=0
MOVL C01607 V=800.0 PL=0
MOVL C01608 V=800.0 PL=0
MOVL C01609 V=800.0 PL=0
MOVL C01610 V=800.0 PL=0
MOVL C01611 V=800.0 PL=0
MOVL C01612 V=800.0 PL=0
MOVL C01613 V=800.0 PL=0
MOVL C01614 V=800.0 PL=0
MOVL C01615 V=800.0 PL=0
MOVL C01616 V=800.0 PL=0
MOVL C01617 V=800.0 PL=0
MOVL C01618 V=800.0 PL=0
MOVL C01619 V=800.0 PL=0
MOVL C01620 V=800.0 PL=0
MOVL C01621 V=800.0 PL=0
MOVL C01622 V=800.0 PL=0
MOVL C01623 V=800.0 PL=0
MOVL C01624 V=800.0 PL=0
MOVL C01625 V=800.0 PL=0
MOVL C01626 V=800.0 PL=0
MOVL C01627 V=800.0 PL=0
MOVL C01628 V=800.0 PL=0
MOVL C01629 V=800.0 PL=0
MOVL C01630 V=800.0 PL=0
MOVL C01631 V=800.0 PL=0
MOVL C01632 V=800.0 PL=0
MOVL C01633 V=800.0 PL=0
MOVL C01634 V=800.0 PL=0
MOVL C01635 V=800.0 PL=0
MOVL C01636 V=800.0 PL=0
MOVL C01637 V=800.0 PL=0
MOVL C01638 V=800.0 PL=0
MOVL C01639 V=800.0 PL=0
MOVL C01640 V=800.0 PL=0
MOVL C01641 V=800.0 PL=0
MOVL C01642 V=800.0 PL=0
MOVL C01643 V=800.0 PL=0
MOVL C01644 V=800.0 PL=0
MOVL C01645 V=800.0 PL=0
MOVL C01646 V=800.0 PL=0
MOVL C01647 V=800.0 PL=0
MOVL C01648 V=800.0 PL=0
MOVL C01649 V=800.0 PL=0
MOVL C01650 V=800.0 PL=0
MOVL C01651 V=800.0 PL=0
MOVL C01652 V=800.0 PL=0
MOVL C01653 V=800.0 PL=0
MOVL C01654 V=800.0 PL=0
MOVL C01655 V=800.0 PL=0
MOVL C01656 V=800.0 PL=0
MOVL C01657 V=800.0 PL=0
MOVL C01658 V=800.0 PL=0
MOVL C01659 V=800.0 PL=0
MOVL C01660 V=800.0 PL=0
MOVL C01661 V=800.0 PL=0
MOVL C01662 V=800.0 PL=0
MOVL C01663 V=800.0 PL=0
MOVL C01664 V=800.0 PL=0
MOVL C01665 V=800.0 PL=0
MOVL C01666 V=800.0 PL=0
MOVL C01667 V=800.0 PL=0
MOVL C01668 V=800.0 PL=0
MOVL C01669 V=800.0 PL=0
MOVL C01670 V=800.0 PL=0
MOVL C01671 V=800.0 PL=0
MOVL C01672 V=800.0 PL=0
MOVL C01673 V=800.0 PL=0
MOVL C01674 V=800.0 PL=0
MOVL C01675 V=800.0 PL=0
MOVL C01676 V=800.0 PL=0
MOVL C01677 V=800.0 PL=0
MOVL C01678 V=800.0 PL=0
MOVL C01679 V=800.0 PL=0
MOVL C01680 V=800.0 PL=0
MOVL C01681 V=800.0 PL=0
MOVL C01682 V=800.0 PL=0
MOVL C01683 V=800.0 PL=0
MOVL C01684 V=800.0 PL=0
MOVL C01685 V=800.0 PL=0
MOVL C01686 V=800.0 PL=0
MOVL C01687 V=800.0 PL=0
MOVL C01688 V=800.0 PL=0
MOVL C01689 V=800.0 PL=0
MOVL C01690 V=800.0 PL=0
MOVL C01691 V=800.0 PL=0
MOVL C01692 V=800.0 PL=0
MOVL C01693 V=800.0 PL=0
MOVL C01694 V=800.0 PL=0
MOVL C01695 V=800.0 PL=0
MOVL C01696 V=800.0 PL=0
MOVL C01697 V=800.0 PL=0
MOVL C01698 V=800.0 PL=0
MOVL C01699 V=800.0 PL=0
MOVL C01700 V=800.0 PL=0
MOVL C01701 V=800.0 PL=0
MOVL C01702 V=800.0 PL=0
MOVL C01703 V=800.0 PL=0
MOVL C01704 V=800.0 PL=0
MOVL C01705 V=800.0 PL=0
MOVL C01706 V=800.0 PL=0
MOVL C01707 V=800.0 PL=0
MOVL C01708 V=800.0 PL=0
MOVL C01709 V=800.0 PL=0
MOVL C01710 V=800.0 PL=0
MOVL C01711 V=800.0 PL=0
MOVL C01712 V=800.0 PL=0
MOVL C01713 V=800.0 PL=0
MOVL C01714 V=800.0 PL=0
MOVL C01715 V=800.0 PL=0
MOVL C01716 V=800.0 PL=0
MOVL C01717 V=800.0 PL=0
MOVL C01718 V=800.0 PL=0
MOVL C01719 V=800.0 PL=0
MOVL C01720 V=800.0 PL=0
MOVL C01721 V=800.0 PL=0
MOVL C01722 V=800.0 PL=0
MOVL C01723 V=800.0 PL=0
MOVL C01724 V=800.0 PL=0
MOVL C01725 V=800.0 PL=0
MOVL C01726 V=800.0 PL=0
MOVL C01727 V=800.0 PL=0
MOVL C01728 V=800.0 PL=0
MOVL C01729 V=800.0 PL=0
MOVL C01730 V=800.0 PL=0
MOVL C01731 V=800.0 PL=0
MOVL C01732 V=800.0 PL=0
MOVL C01733 V=800.0 PL=0
MOVL C01734 V=800.0 PL=0
MOVL C01735 V=800.0 PL=0
MOVL C01736 V=800.0 PL=0
MOVL C01737 V=800.0 PL=0
MOVL C01738 V=800.0 PL=0
MOVL C01739 V=800.0 PL=0
MOVL C01740 V=800.0 PL=0
MOVL C01741 V=800.0 PL=0
MOVL C01742 V=800.0 PL=0
MOVL C01743 V=800.0 PL=0
MOVL C01744 V=800.0 PL=0
MOVL C01745 V=800.0 PL=0
MOVL C01746 V=800.0 PL=0
MOVL C01747 V=800.0 PL=0
MOVL C01748 V=800.0 PL=0
MOVL C01749 V=800.0 PL=0
MOVL C01750 V=800.0 PL=0
MOVL C01751 V=800.0 PL=0
MOVL C01752 V=800.0 PL=0
MOVL C01753 V=800.0 PL=0
MOVL C01754 V=800.0 PL=0
MOVL C01755 V=800.0 PL=0
MOVL C01756 V=800.0 PL=0
MOVL C01757 V=800.0 PL=0
MOVL C01758 V=800.0 PL=0
MOVL C01759 V=800.0 PL=0
MOVL C01760 V=800.0 PL=0
MOVL C01761 V=800.0 PL=0
MOVL C01762 V=800.0 PL=0
MOVL C01763 V=800.0 PL=0
MOVL C01764 V=800.0 PL=0
MOVL C01765 V=800.0 PL=0
MOVL C01766 V=800.0 PL=0
MOVL C01767 V=800.0 PL=0
MOVL C01768 V=800.0 PL=0
MOVL C01769 V=800.0 PL=0
MOVL C01770 V=800.0 PL=0
MOVL C01771 V=800.0 PL=0
MOVL C01772 V=800.0 PL=0
MOVL C01773 V=800.0 PL=0
MOVL C01774 V=800.0 PL=0
MOVL C01775 V=800.0 PL=0
MOVL C01776 V=800.0 PL=0
MOVL C01777 V=800.0 PL=0
MOVL C01778 V=800.0 PL=0
MOVL C01779 V=800.0 PL=0
MOVL C01780 V=800.0 PL=0
MOVL C01781 V=800.0 PL=0
MOVL C01782 V=800.0 PL=0
MOVL C01783 V=800.0 PL=0
MOVL C01784 V=800.0 PL=0
MOVL C01785 V=800.0 PL=0
MOVL C01786 V=800.0 PL=0
MOVL C01787 V=800.0 PL=0
MOVL C01788 V=800.0 PL=0
MOVL C01789 V=800.0 PL=0
MOVL C01790 V=800.0 PL=0
MOVL C01791 V=800.0 PL=0
MOVL C01792 V=800.0 PL=0
MOVL C01793 V=800.0 PL=0
MOVL C01794 V=800.0 PL=0
MOVL C01795 V=800.0 PL=0
MOVL C01796 V=800.0 PL=0
MOVL C01797 V=800.0 PL=0
MOVL C01798 V=800.0 PL=0
MOVL C01799 V=800.0 PL=0
MOVL C01800 V=800.0 PL=0
MOVL C01801 V=800.0 PL=0
MOVL C01802 V=800.0 PL=0
MOVL C01803 V=800.0 PL=0
MOVL C01804 V=800.0 PL=0
MOVL C01805 V=800.0 PL=0
MOVL C01806 V=800.0 PL=0
MOVL C01807 V=800.0 PL=0
MOVL C01808 V=800.0 PL=0
MOVL C01809 V=800.0 PL=0
MOVL C01810 V=800.0 PL=0
MOVL C01811 V=800.0 PL=0
MOVL C01812 V=800.0 PL=0
MOVL C01813 V=800.0 PL=0
MOVL C01814 V=800.0 PL=0
MOVL C01815 V=800.0 PL=0
MOVL C01816 V=800.0 PL=0
MOVL C01817 V=800.0 PL=0
MOVL C01818 V=800.0 PL=0
MOVL C01819 V=800.0 PL=0
MOVL C01820 V=800.0 PL=0
MOVL C01821 V=800.0 PL=0
MOVL C01822 V=800.0 PL=0
MOVL C01823 V=800.0 PL=0
MOVL C01824 V=800.0 PL=0
MOVL C01825 V=800.0 PL=0
MOVL C01826 V=800.0 PL=0
MOVL C01827 V=800.0 PL=0
MOVL C01828 V=800.0 PL=0
MOVL C01829 V=800.0 PL=0
MOVL C01830 V=800.0 PL=0
MOVL C01831 V=800.0 PL=0
MOVL C01832 V=800.0 PL=0
MOVL C01833 V=800.0 PL=0
MOVL C01834 V=800.0 PL=0
MOVL C01835 V=800.0 PL=0
MOVL C01836 V=800.0 PL=0
MOVL C01837 V=800.0 PL=0
MOVL C01838 V=800.0 PL=0
MOVL C01839 V=800.0 PL=0
MOVL C01840 V=800.0 PL=0
MOVL C01841 V=800.0 PL=0
MOVL C01842 V=800.0 PL=0
MOVL C01843 V=800.0 PL=0
MOVL C01844 V=800.0 PL=0
MOVL C01845 V=800.0 PL=0
MOVL C01846 V=800.0 PL=0
MOVL C01847 V=800.0 PL=0
MOVL C01848 V=800.0 PL=0
MOVL C01849 V=800.0 PL=0
MOVL C01850 V=800.0 PL=0
MOVL C01851 V=800.0 PL=0
MOVL C01852 V=800.0 PL=0
MOVL C01853 V=800.0 PL=0
MOVL C01854 V=800.0 PL=0
MOVL C01855 V=800.0 PL=0
MOVL C01856 V=800.0 PL=0
MOVL C01857 V=800.0 PL=0
MOVL C01858 V=800.0 PL=0
MOVL C01859 V=800.0 PL=0
MOVL C01860 V=800.0 PL=0
MOVL C01861 V=800.0 PL=0
MOVL C01862 V=800.0 PL=0
MOVL C01863 V=800.0 PL=0
MOVL C01864 V=800.0 PL=0
MOVL C01865 V=800.0 PL=0
MOVL C01866 V=800.0 PL=0
MOVL C01867 V=800.0 PL=0
MOVL C01868 V=800.0 PL=0
MOVL C01869 V=800.0 PL=0
MOVL C01870 V=800.0 PL=0
MOVL C01871 V=800.0 PL=0
MOVL C01872 V=800.0 PL=0
MOVL C01873 V=800.0 PL=0
MOVL C01874 V=800.0 PL=0
MOVL C01875 V=800.0 PL=0
MOVL C01876 V=800.0 PL=0
MOVL C01877 V=800.0 PL=0
MOVL C01878 V=800.0 PL=0
MOVL C01879 V=800.0 PL=0
MOVL C01880 V=800.0 PL=0
MOVL C01881 V=800.0 PL=0
MOVL C01882 V=800.0 PL=0
MOVL C01883 V=800.0 PL=0
MOVL C01884 V=800.0 PL=0
MOVL C01885 V=800.0 PL=0
MOVL C01886 V=800.0 PL=0
MOVL C01887 V=800.0 PL=0
MOVL C01888 V=800.0 PL=0
MOVL C01889 V=800.0 PL=0
MOVL C01890 V=800.0 PL=0
MOVL C01891 V=800.0 PL=0
MOVL C01892 V=800.0 PL=0
MOVL C01893 V=800.0 PL=0
MOVL C01894 V=800.0 PL=0
MOVL C01895 V=800.0 PL=0
MOVL C01896 V=800.0 PL=0
MOVL C01897 V=800.0 PL=0
MOVL C01898 V=800.0 PL=0
MOVL C01899 V=800.0 PL=0
MOVL C01900 V=800.0 PL=0
MOVL C01901 V=800.0 PL=0
MOVL C01902 V=800.0 PL=0
MOVL C01903 V=800.0 PL=0
MOVL C01904 V=800.0 PL=0
MOVL C01905 V=800.0 PL=0
MOVL C01906 V=800.0 PL=0
MOVL C01907 V=800.0 PL=0
MOVL C01908 V=800.0 PL=0
MOVL C01909 V=800.0 PL=0
MOVL C01910 V=800.0 PL=0
MOVL C01911 V=800.0 PL=0
MOVL C01912 V=800.0 PL=0
MOVL C01913 V=800.0 PL=0
MOVL C01914 V=800.0 PL=0
MOVL C01915 V=800.0 PL=0
MOVL C01916 V=800.0 PL=0
MOVL C01917 V=800.0 PL=0
MOVL C01918 V=800.0 PL=0
MOVL C01919 V=800.0 PL=0
MOVL C01920 V=800.0 PL=0
MOVL C01921 V=800.0 PL=0
MOVL C01922 V=800.0 PL=0
MOVL C01923 V=800.0 PL=0
MOVL C01924 V=800.0 PL=0
MOVL C01925 V=800.0 PL=0
MOVL C01926 V=800.0 PL=0
MOVL C01927 V=800.0 PL=0
MOVL C01928 V=800.0 PL=0
MOVL C01929 V=800.0 PL=0
MOVL C01930 V=800.0 PL=0
MOVL C01931 V=800.0 PL=0
MOVL C01932 V=800.0 PL=0
MOVL C01933 V=800.0 PL=0
MOVL C01934 V=800.0 PL=0
MOVL C01935 V=800.0 PL=0
MOVL C01936 V=800.0 PL=0
MOVL C01937 V=800.0 PL=0
MOVL C01938 V=800.0 PL=0
MOVL C01939 V=800.0 PL=0
MOVL C01940 V=800.0 PL=0
MOVL C01941 V=800.0 PL=0
MOVL C01942 V=800.0 PL=0
MOVL C01943 V=800.0 PL=0
MOVL C01944 V=800.0 PL=0
MOVL C01945 V=800.0 PL=0
MOVL C01946 V=800.0 PL=0
MOVL C01947 V=800.0 PL=0
MOVL C01948 V=800.0 PL=0
MOVL C01949 V=800.0 PL=0
MOVL C01950 V=800.0 PL=0
MOVL C01951 V=800.0 PL=0
MOVL C01952 V=800.0 PL=0
MOVL C01953 V=800.0 PL=0
MOVL C01954 V=800.0 PL=0
MOVL C01955 V=800.0 PL=0
MOVL C01956 V=800.0 PL=0
MOVL C01957 V=800.0 PL=0
MOVL C01958 V=800.0 PL=0
MOVL C01959 V=800.0 PL=0
MOVL C01960 V=800.0 PL=0
MOVL C01961 V=800.0 PL=0
MOVL C01962 V=800.0 PL=0
MOVL C01963 V=800.0 PL=0
MOVL C01964 V=800.0 PL=0
MOVL C01965 V=800.0 PL=0
MOVL C01966 V=800.0 PL=0
MOVL C01967 V=800.0 PL=0
MOVL C01968 V=800.0 PL=0
MOVL C01969 V=800.0 PL=0
MOVL C01970 V=800.0 PL=0
MOVL C01971 V=800.0 PL=0
MOVL C01972 V=800.0 PL=0
MOVL C01973 V=800.0 PL=0
MOVL C01974 V=800.0 PL=0
MOVL C01975 V=800.0 PL=0
MOVL C01976 V=800.0 PL=0
MOVL C01977 V=800.0 PL=0
MOVL C01978 V=800.0 PL=0
MOVL C01979 V=800.0 PL=0
MOVL C01980 V=800.0 PL=0
MOVL C01981 V=800.0 PL=0
MOVL C01982 V=800.0 PL=0
MOVL C01983 V=800.0 PL=0
MOVL C01984 V=800.0 PL=0
MOVL C01985 V=800.0 PL=0
MOVL C01986 V=800.0 PL=0
MOVL C01987 V=800.0 PL=0
MOVL C01988 V=800.0 PL=0
MOVL C01989 V=800.0 PL=0
MOVL C01990 V=800.0 PL=0
MOVL C01991 V=800.0 PL=0
MOVL C01992 V=800.0 PL=0
MOVL C01993 V=800.0 PL=0
MOVL C01994 V=800.0 PL=0
MOVL C01995 V=800.0 PL=0
MOVL C01996 V=800.0 PL=0
MOVL C01997 V=800.0 PL=0
MOVL C01998 V=800.0 PL=0
MOVL C01999 V=800.0 PL=0
MOVL C02000 V=800.0 PL=0
MOVL C02001 V=800.0 PL=0
MOVL C02002 V=800.0 PL=0
MOVL C02003 V=800.0 PL=0
MOVL C02004 V=800.0 PL=0
MOVL C02005 V=800.0 PL=0
MOVL C02006 V=800.0 PL=0
MOVL C02007 V=800.0 PL=0
MOVL C02008 V=800.0 PL=0
MOVL C02009 V=800.0 PL=0
MOVL C02010 V=800.0 PL=0
MOVL C02011 V=800.0 PL=0
MOVL C02012 V=800.0 PL=0
MOVL C02013 V=800.0 PL=0
MOVL C02014 V=800.0 PL=0
MOVL C02015 V=800.0 PL=0
MOVL C02016 V=800.0 PL=0
MOVL C02017 V=800.0 PL=0
MOVL C02018 V=800.0 PL=0
MOVL C02019 V=800.0 PL=0
MOVL C02020 V=800.0 PL=0
MOVL C02021 V=800.0 PL=0
MOVL C02022 V=800.0 PL=0
MOVL C02023 V=800.0 PL=0
MOVL C02024 V=800.0 PL=0
MOVL C02025 V=800.0 PL=0
MOVL C02026 V=800.0 PL=0
MOVL C02027 V=800.0 PL=0
MOVL C02028 V=800.0 PL=0
MOVL C02029 V=800.0 PL=0
MOVL C02030 V=800.0 PL=0
MOVL C02031 V=800.0 PL=0
MOVL C02032 V=800.0 PL=0
MOVL C02033 V=800.0 PL=0
MOVL C02034 V=800.0 PL=0
MOVL C02035 V=800.0 PL=0
MOVL C02036 V=800.0 PL=0
MOVL C02037 V=800.0 PL=0
MOVL C02038 V=800.0 PL=0
MOVL C02039 V=800.0 PL=0
MOVL C02040 V=800.0 PL=0
MOVL C02041 V=800.0 PL=0
MOVL C02042 V=800.0 PL=0
MOVL C02043 V=800.0 PL=0
MOVL C02044 V=800.0 PL=0
MOVL C02045 V=800.0 PL=0
MOVL C02046 V=800.0 PL=0
MOVL C02047 V=800.0 PL=0
MOVL C02048 V=800.0 PL=0
MOVL C02049 V=800.0 PL=0
MOVL C02050 V=800.0 PL=0
MOVL C02051 V=800.0 PL=0
MOVL C02052 V=800.0 PL=0
MOVL C02053 V=800.0 PL=0
